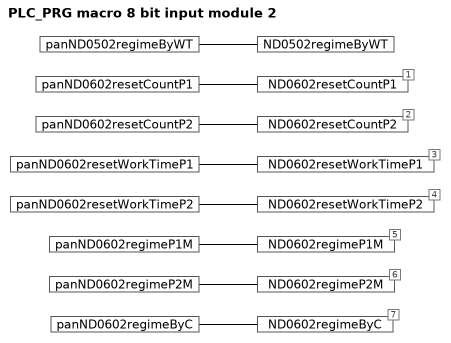
[picture p72: PLC_PRG macro 8 bit input module 2 (CFC)]
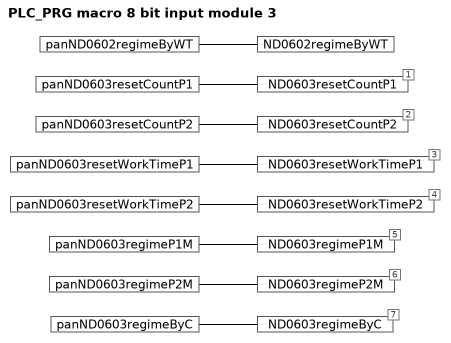
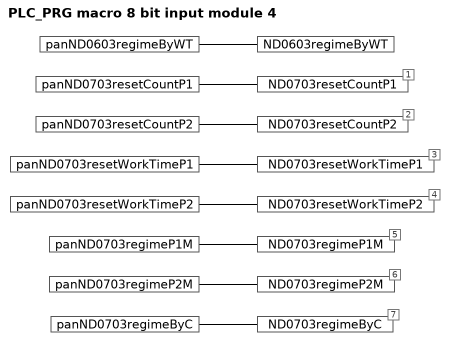
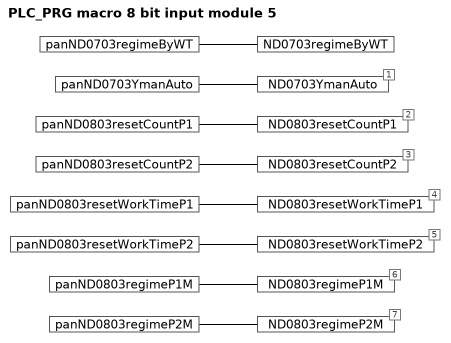
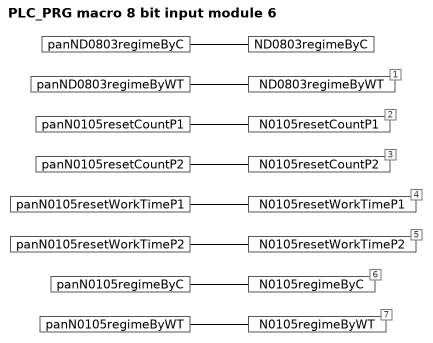
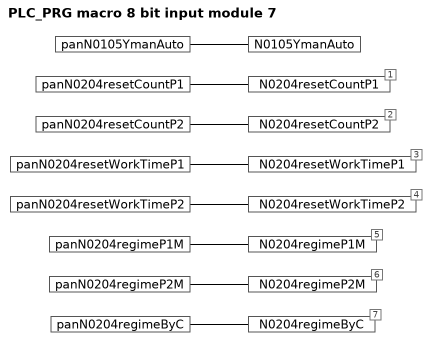
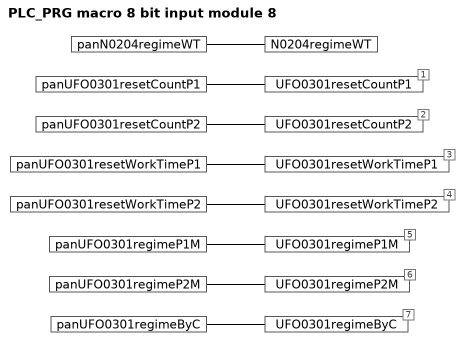
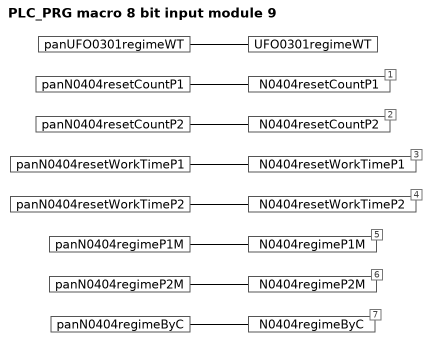
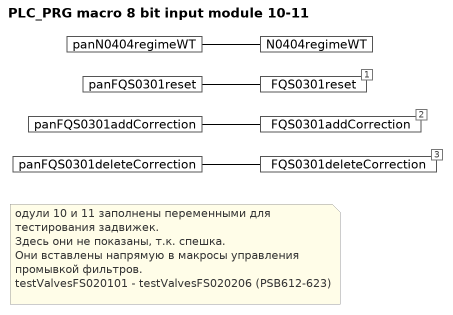
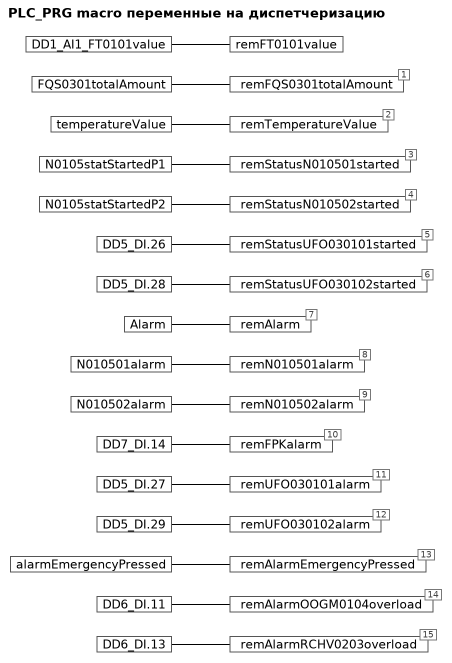
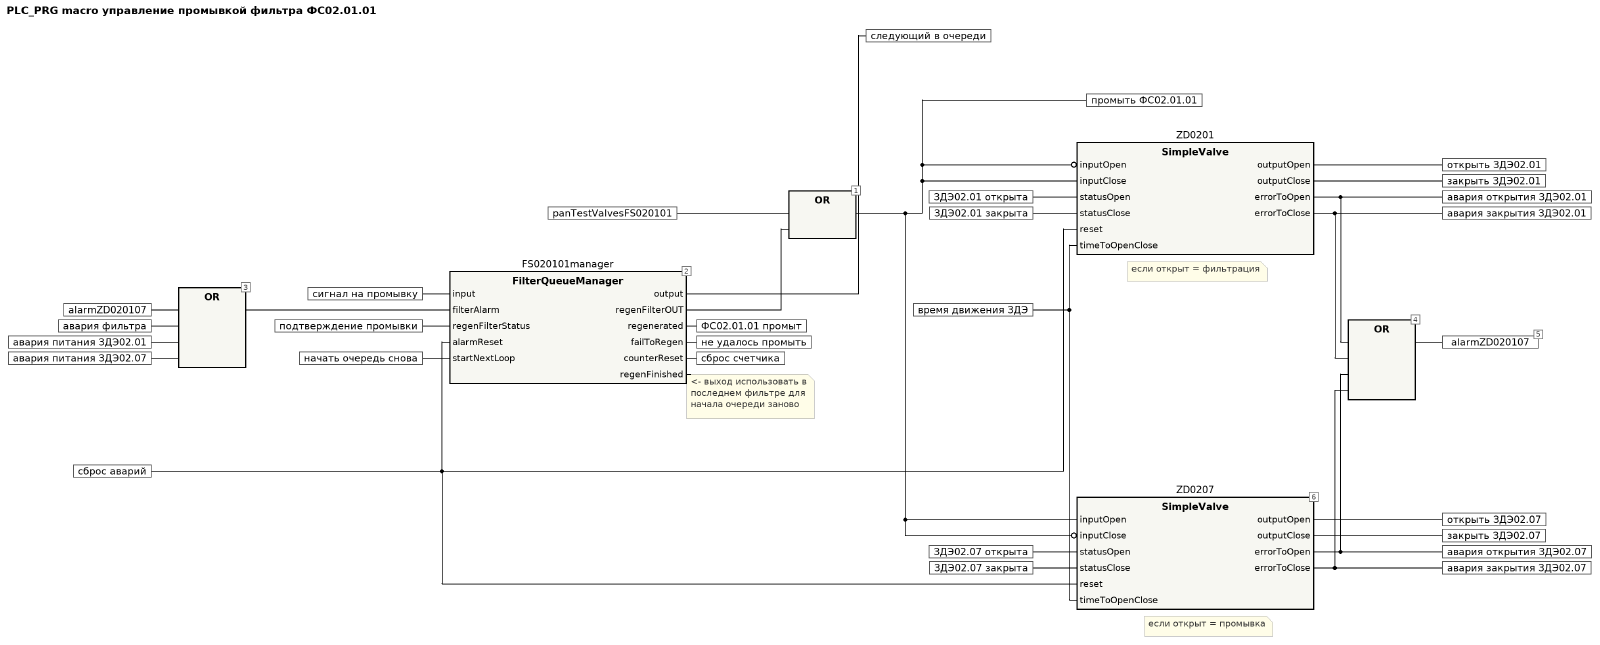
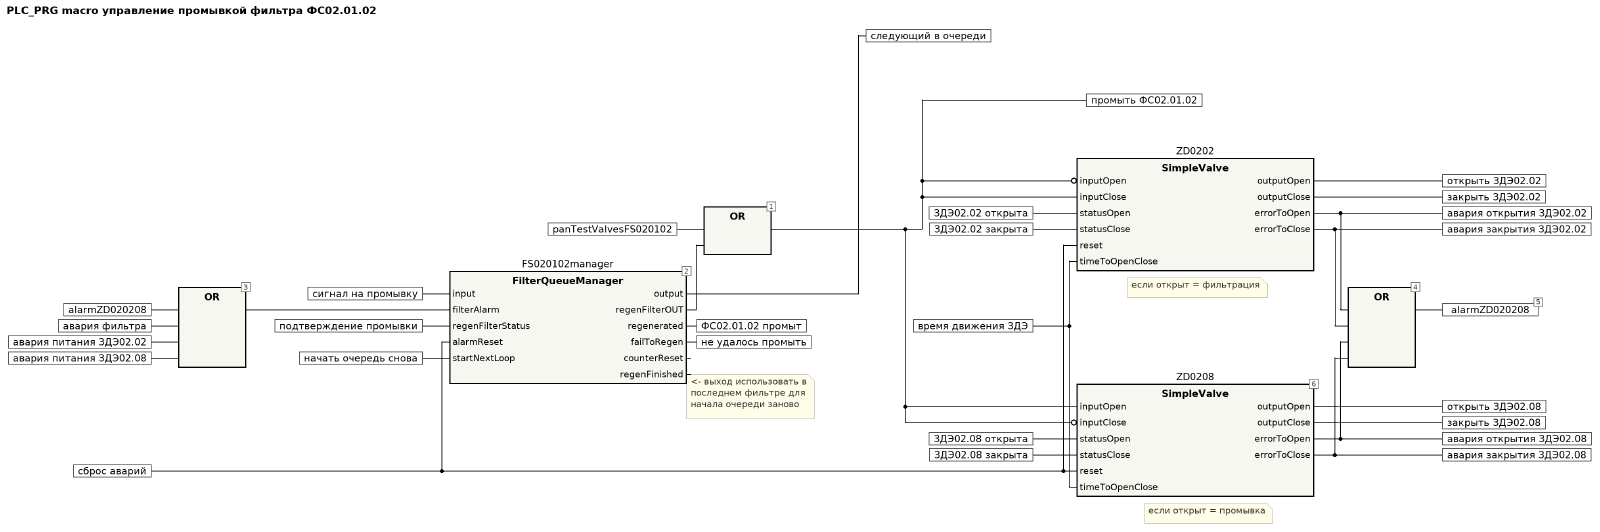
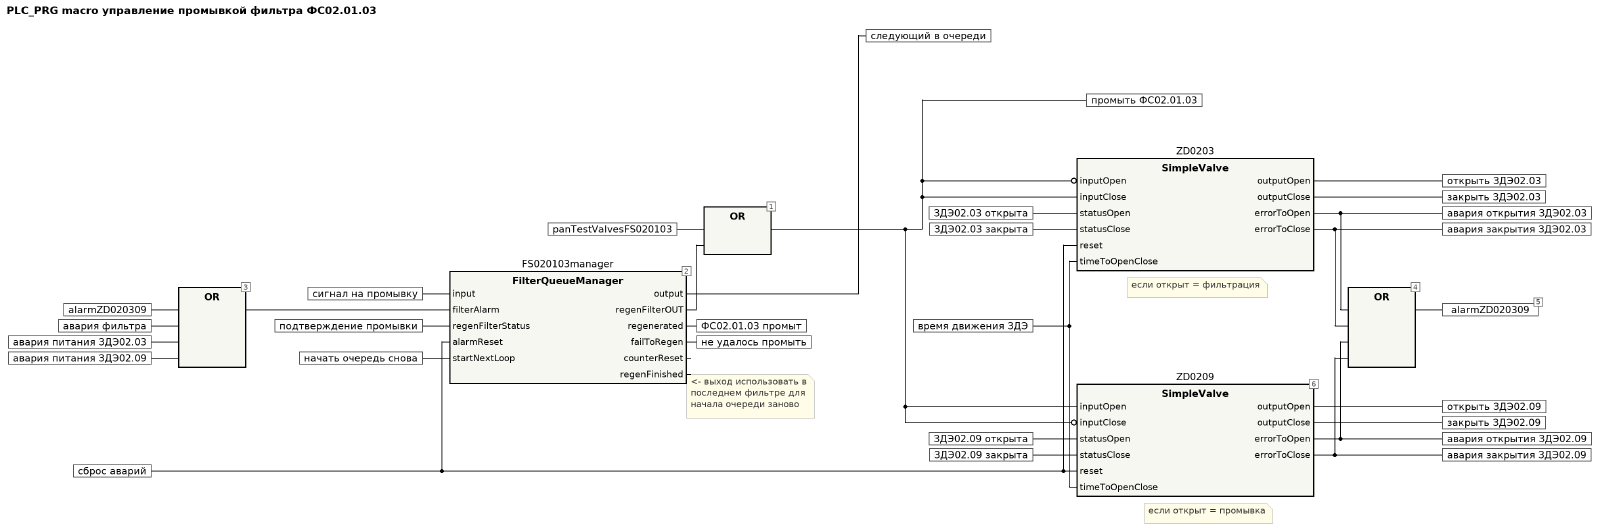
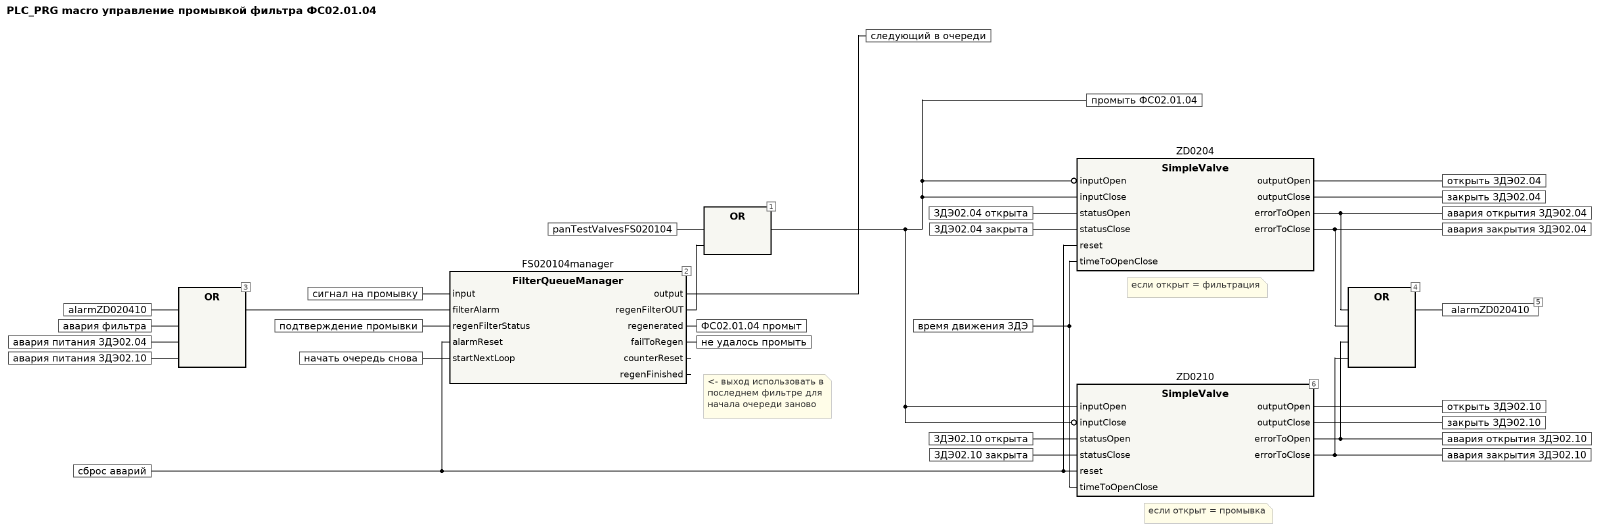
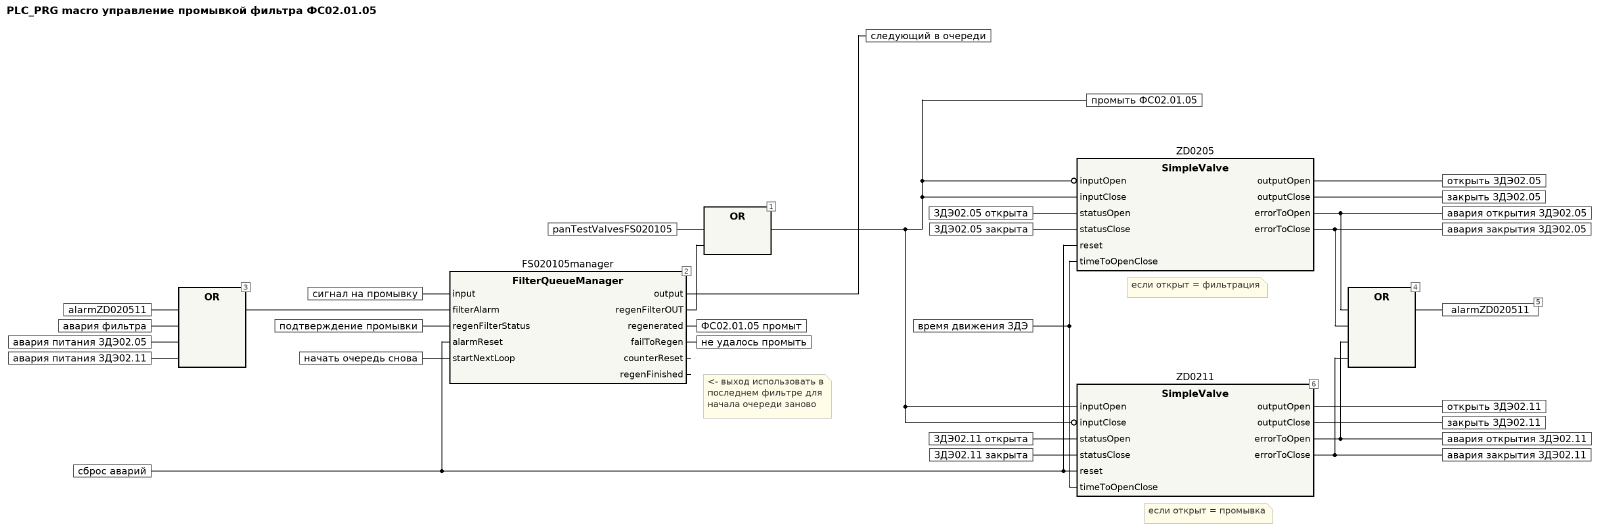
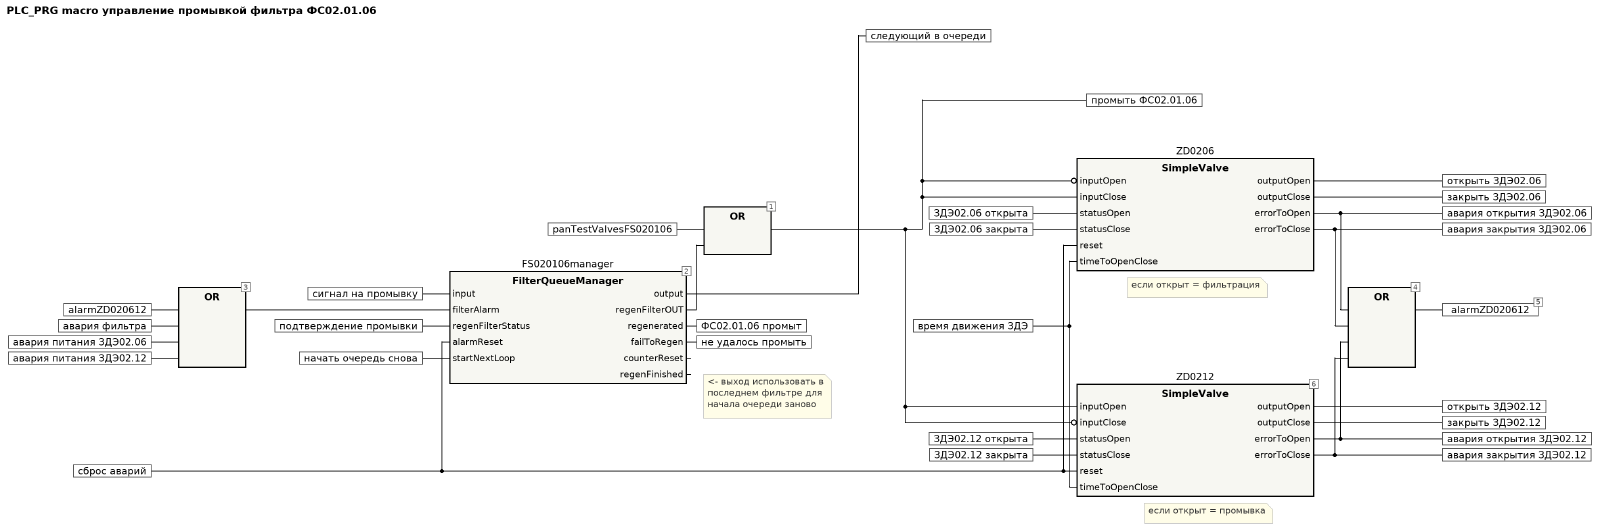
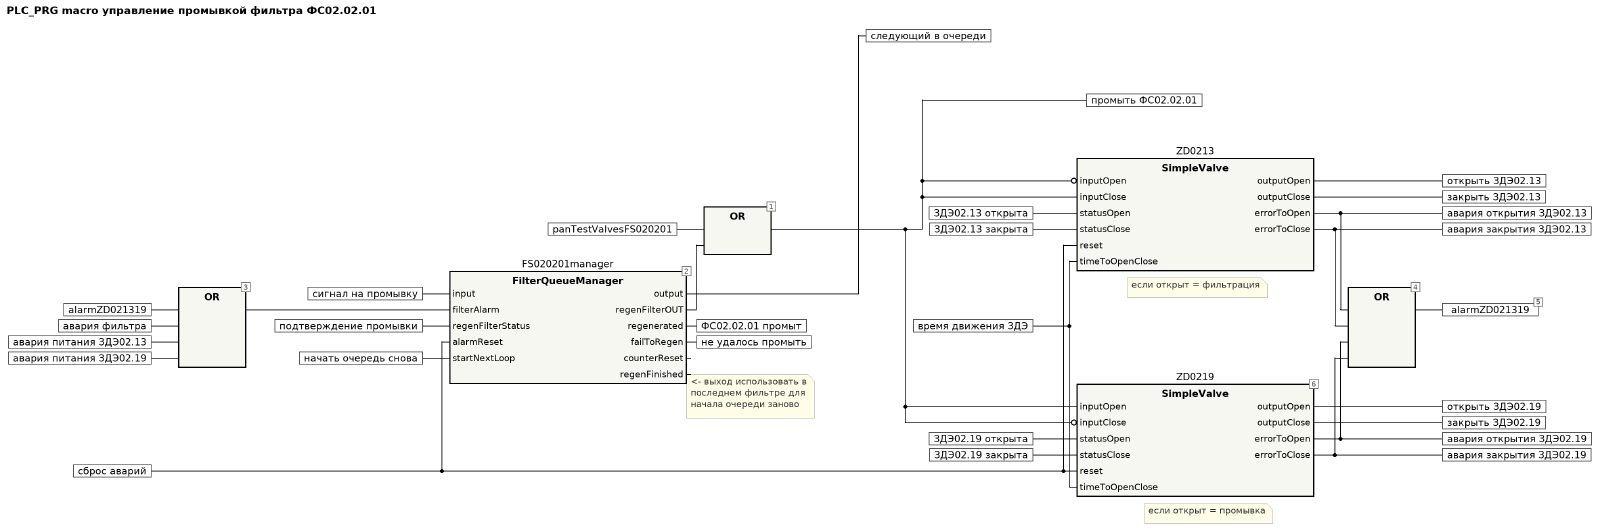
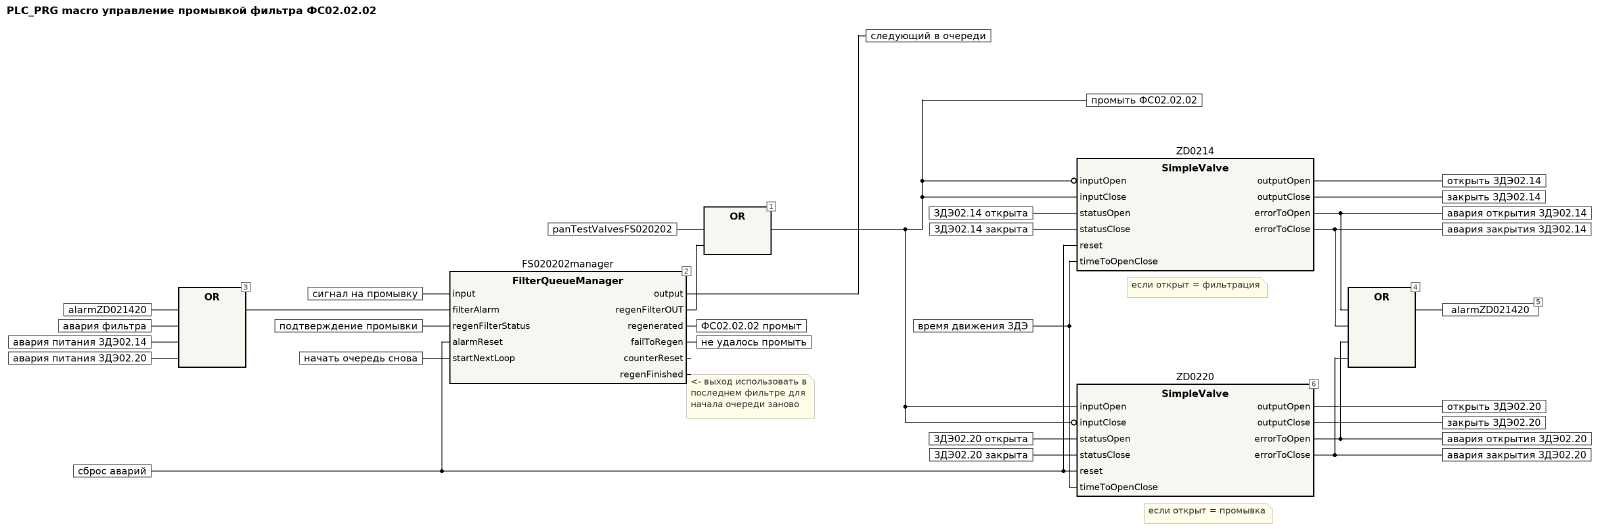
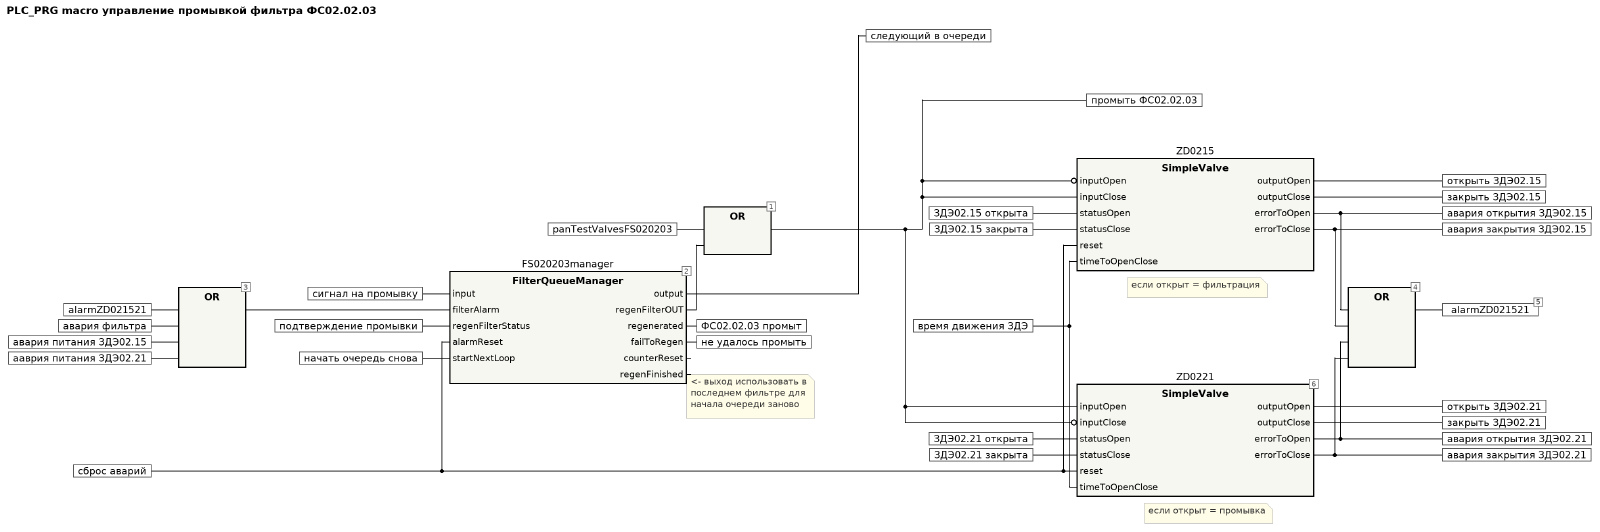
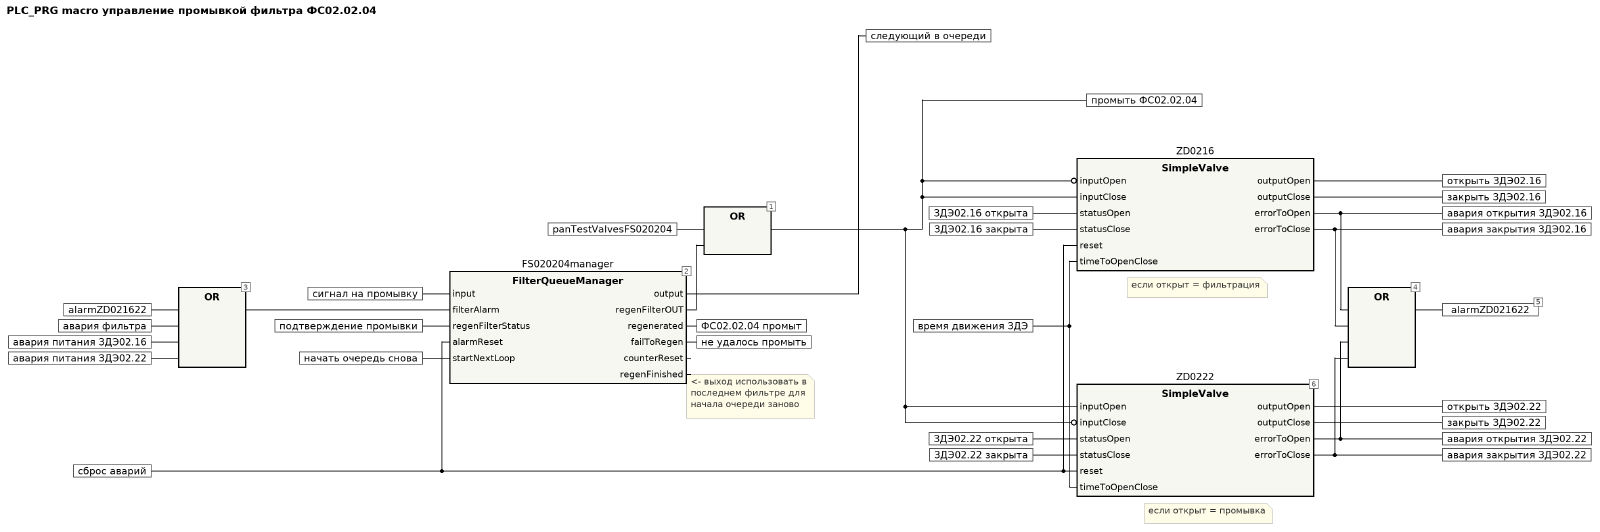
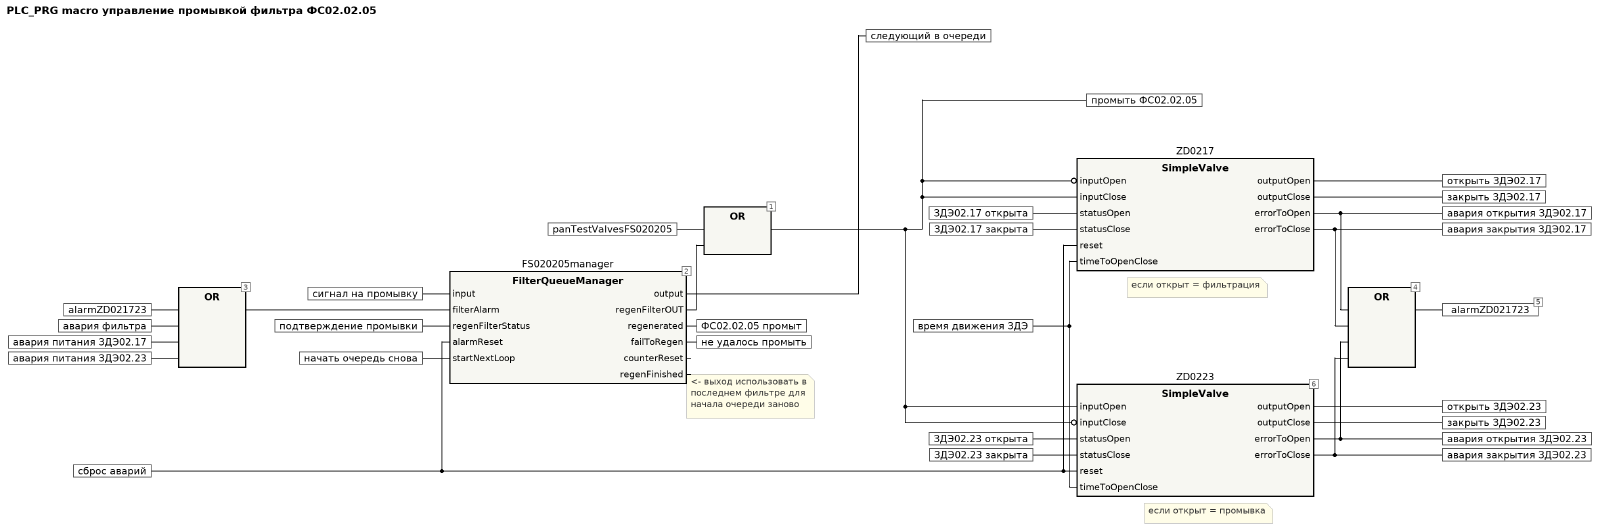
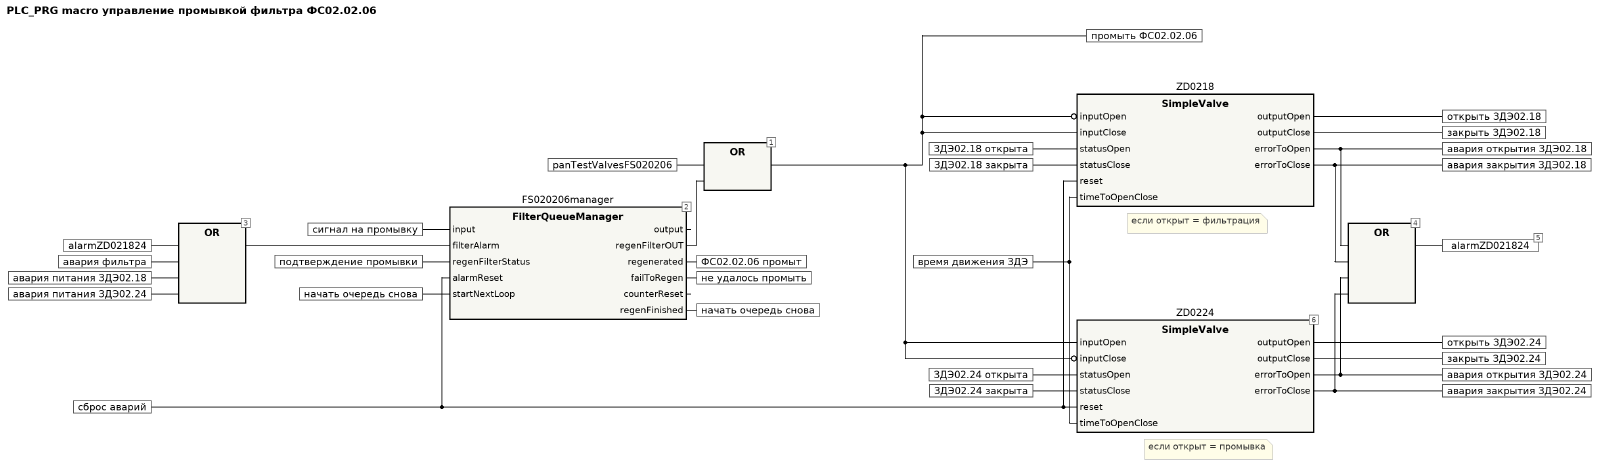
_CFC_ (* Continuous Function Chart, elements in execution order *)
(* 0 = перелив *)
(* авария обоих УФО, если проблемы / открытия/закрытия на одной из задвижек *)
(* авария питания ЗДЭ03.02 *)
(* авария питания ЗДЭ03.01 *)
(* статус-пуск Н01.05/02 *)
(* вкл КМ3 *)
(* Статус ПУСК / ЧРП Н01.05 *)
(* статус-пуск Н01.05/01 *)
(* вкл КМ2 *)
(* контроль обрыва или ошибок модулей в сети ПЛК *)
(* LSA01.02 перелив ОГМ01.04 *)
(* Нажат аварийный стоп. *)
(* авария сети (РКФ) *)
(* разрешение работы КНС / 1 = разрешено *)
(* Нажат аварийный стоп. *)
(* Блок управления разрешением работы КНС *)
(* авария сети (РКФ) *)
(* Авария питания клапанов КЭМ. *)
(* Авария питания розеток / управл.клапанов фильтров. *)
(* авария КНС *)
(* блок подачи сигнала на промывку *)
(* суммируем каждую секунду значение / мгновенного расхода в кубометрах в секунду *)
(* преобразуем расход из / кубометров в час в / кубометры в секунду *)
(* если есть расход / (больше нуля) *)
(* выдает импульс / каждую секунду *)
(* здесь мгновенный расход / в кубометрах в час (FT01.02) *)
(* Авария Н02.04/01 (0=авария) *)
(* Авария Н02.04/02 (0=авария) *)
(* промывка ФС02.01/06 *)
(* промывка ФС02.01/05 *)
(* промывка ФС02.01/04 *)
(* промывка ФС02.01/03 *)
(* промывка ФС02.01/02 *)
(* промывка ФС02.01/01 *)
(* пуск/стоп НД08.03/01 *)
(* пуск/стоп НД08.03/02 *)
(* пуск/стоп НД06.03/01 *)
(* пуск/стоп НД06.03/02 *)
(* пуск/стоп НД06.02/01 *)
(* пуск/стоп НД06.02/02 *)
(* пуск/стоп НД08.04 *)
(* пуск/стоп НД07.03/01 *)
(* пуск/стоп НД07.03/02 *)
(* авария М08.02 (УПФ) *)
(* авария М07.02 (УПЩ) *)
(* авария М06.04 (УПК) *)
(* работа М08.02 (УПФ) *)
(* работа М07.02 (УПЩ) *)
(* работа М06.04 (УПК) *)
(* Контроль, если УФО включили вручную, / а потока при этом нет. *)
(* авария УФО03.01/02 *)
(* работа УФО03.01/02 *)
(* авария УФО03.01/01 *)
(* Для подачи предостережения на пульте / оператора (при необходимости), а также / сигнализации лампой АВАРИЯ. *)
(* работа УФО03.01/01 *)
(* авария УФО03.01/02 *)
(* авария УФО03.01/01 *)
(* авария Н04.04/01 *)
(* авария Н04.04/02 *)
(* время контроля старта ФПК (по умолч.=3мин) *)
(* время работы ФПК после спада сигнала датч.осадка *)
(* запуск фильтрации *)
(* Защита от сухого хода насоса ФПК *)
(* датчик уровня осадка *)
(* Давление на входе ФПК (0...16 бар) *)
(* авария ФПК *)
(* подающий насос ФПК работает *)
(* ФПК готов к приему *)
(* ФПК не запустился *)
(* рН-метр QE01.02 на входе, / диапазон 0...14 *)
(* авария входа рН-метра QE01.01 *)
(* авария входа расходомера FT01.02 *)
(* расходомер FT01.01 на входе, / диапазон 0...600куб/час *)
(* авария НД08.04 *)
(* управление 4...20мА НД08.03/01 *)
(* пуск/стоп НД08.03/01 *)
(* пуск/стоп НД08.03/02 *)
(* управление 4...20мА НД08.03/02 *)
(* авария привода НД08.03/01 *)
(* авария привода НД08.03/02 *)
(* авария НД07.03/01 *)
(* авария НД07.03/02 *)
(* управление 4...20мА НД07.03/01 *)
(* управление 4...20мА НД07.03/02 *)
(* пуск/стоп НД07.03/01 *)
(* пуск/стоп НД07.03/02 *)
(* авария НД07.03/01 *)
(* авария НД07.03/02 *)
(* авария НД06.03/01 *)
(* авария НД06.03/02 *)
(* авария НД06.02/01 *)
(* авария НД06.02/02 *)
(* управление 4...20мА НД06.03/01 *)
(* пуск/стоп НД06.03/01 *)
(* пуск/стоп НД06.03/02 *)
(* управление 4...20мА НД06.03/02 *)
(* авария НД06.03/01 *)
(* авария НД06.03/02 *)
(* управление 4...20мА НД06.02/01 *)
(* пуск/стоп НД06.02/01 *)
(* пуск/стоп НД06.02/02 *)
(* управление 4...20мА НД06.02/02 *)
(* авария НД06.02/01 *)
(* авария НД06.02/02 *)
(* ошибка блока дозирования НД05.02 *)
(* авария входа датчика температуры *)
(* лампа АВАРИЯ *)
(* датчик температуры в помещении / (метран) диапазон: 0...+100С *)
(* управление 4...20мА НД05.02/01 *)
(* пуск/стоп НД05.02/01 *)
(* авария НД05.02/01 *)
(* авария НД05.02/02 *)
(* пуск/стоп НД05.02/02 *)
(* управление 4...20мА НД05.02/02 *)
(* АВАРИИ *)
(* авария привода НД08.03/01 *)
(* авария привода НД08.03/02 *)
(* авария НД08.04 *)
(* насос Н04.01 работает *)
(* пуск/стоп НД08.04 *)
(* управление 4...20мА НД08.04 *)
(* авария входа расходомера FT01.01 *)
(* расходомер FT01.02 на входе, / диапазон 0...600куб/час *)
(* рН-метр QE01.01 на входе, / диапазон 0...14 *)
(* авария входа рН-метра QE01.02 *)
(* сухой ход НД08.03/01 *)
(* сухой ход НД08.03/02 *)
(* сухой ход НД08.03/01 *)
(* сухой ход НД08.03/02 *)
(* LSA01.02 перелив ОГМ01.04 *)
(* Инициализирует требуемые булевые переменные / в момент старта выполнения программы. *)
(* Статус ПУСК ЧРП Н01.05 *)
(* LS01.03 - рабочий верхний уровень ОГМ01.04 автоматический пуск 01.05 *)
(* LS01.04 - нижний уровень ОГМ01.04, сухой ход Н01.05 *)
(* SA1 Ручной выбор Н01.05/01 = главный *)
(* SA1 Ручной выбор Н01.05/02 = главный *)
(* Стоп  Н01.05 (сброс самоподхвата реле) *)
(* время на создание потока *)
(* Пуск  Н01.05 *)
(* КМ1 питание ЧРП *)
(* КМ2 питание насоса 1 *)
(* КМ3 питание насоса 2 *)
(* Авария ЧРП Н01.05 *)
(* термоконтакт Н01.05/01 *)
(* термоконтакт Н01.05/02 *)
(* авария питания ЗДЭ02.25 *)
(* LSА02.01 Перелив РЧВ02.03 *)
(* Давление на входе ФПК / 0...16 бар (мах допуст.10) *)
(* Авария входа AI6 ПЛК, давл.ФПК *)
(* авария ФПК *)
(* Открыть КШЭ04.01 *)
(* статус КШЭ04.01 открыт *)
(* Закрыть КШЭ04.01 *)
(* статус КШЭ04.01 закрыт *)
(* подающий насос ФПК работает *)
(* стоп Н04.04 *)
(* пуск Н04.04/02 *)
(* пуск Н04.04/01 *)
(* авт.пуск Н04.04 *)
(* сухой ход Н04.04, 0=защита *)
(* авария Н04.04/01, 0=авария *)
(* авария Н04.04/02, 0=авария *)
(* импульсный расходомер *)
(* Авария Н02.04/01 (0=авария) *)
(* Авария Н02.04/02 (0=авария) *)
(* промывка ФС02.02/06 *)
(* промывка ФС02.02/05 *)
(* промывка ФС02.02/04 *)
(* промывка ФС02.02/03 *)
(* промывка ФС02.02/02 *)
(* промывка ФС02.02/01 *)
(* Клапан КЭМ05.01 открыт. *)
(* Клапан КЭМ06.01 открыт. *)
(* Клапан КЭМ07.01 открыт. *)
(* Клапан КЭМ08.01 открыт. *)
(* Сухой ход Н02.04 (LS02.03) 0=сух.ход *)
(* Стоп Н02.04 *)
(* Пуск Н02.04/01 *)
(* Пуск Н02.04/02 *)
(* текущий объем *)
(* заданный до промывки объем *)
(* 0=авария *)
(* авария (при 0) ФС02.01/06 *)
(* авария (при 0) ФС02.01/05 *)
(* авария (при 0) ФС02.01/04 *)
(* авария (при 0) ФС02.01/03 *)
(* авария (при 0) ФС02.01/02 *)
(* авария (при 0) ФС02.01/01 *)
(* авария (при 0) ФС02.02/06 *)
(* авария (при 0) ФС02.02/05 *)
(* авария (при 0) ФС02.02/04 *)
(* авария (при 0) ФС02.02/03 *)
(* авария (при 0) ФС02.02/02 *)
(* авария (при 0) ФС02.02/01 *)
(* сброс счетчика стоков до следующей промывки *)
(* подсчет общего объема стоков, прошедшего через расходомер FT01.02 *)
(* очередь передается на 2 ступень *)
(* авария питания ЗДЭ02.01 *)
(* авария питания ЗДЭ02.02 *)
(* авария питания ЗДЭ02.03 *)
(* авария питания ЗДЭ02.04 *)
(* авария питания ЗДЭ02.05 *)
(* авария питания ЗДЭ02.06 *)
(* авария питания ЗДЭ02.07 *)
(* авария питания ЗДЭ02.08 *)
(* авария питания ЗДЭ02.09 *)
(* авария питания ЗДЭ02.10 *)
(* авария питания ЗДЭ02.11 *)
(* авария питания ЗДЭ02.12 *)
(* авария питания ЗДЭ02.13 *)
(* авария питания ЗДЭ02.14 *)
(* авария питания ЗДЭ02.15 *)
(* авария питания ЗДЭ02.16 *)
(* авария питания ЗДЭ02.17 *)
(* авария питания ЗДЭ02.18 *)
(* авария питания ЗДЭ02.19 *)
(* авария питания ЗДЭ02.20 *)
(* авария питания ЗДЭ02.21 *)
(* авария питания ЗДЭ02.22 *)
(* авария питания ЗДЭ02.23 *)
(* авария питания ЗДЭ02.24 *)
(* инвертирование сигнала, чтобы все аварии / обозначались как 1 (TRUE) *)
(* авария НД05.02/01 *)
(* авария НД05.02/02 *)
(* авария питания КШЭ04.01 *)
(* 1=открыть; 0 = закрыть *)
(* в этом макросе лежит управление режимом тестирования задвижек ЗДЭ03 / Тестирование запрещает автоматический запуск УФО от ПЛК *)
#0 rTrigStartInitializer:R_TRIG(CLK: TRUE)
#1 startInitializer <= #0.Q
#2 MACRO контроль температуры в помещении(pin 1 "вход датчика температуры": DD1_AI0, pin 2 "минимально допустимая температура в помещении": maxTemperature, pin 3 "максимально допустимая температура в помещении": minTemperature)
	(* задаем границы допустимой температуры в помещении / проверяем что измеренное значение в заданном диапазоне *)
	(* не смотрим конкретный тип ошибки / (работает не точно, обрыв определяет как слишком маленькое значение) / если не равно 0 - значит на входе ошибка *)
	#3 DD1_AI0_temperature:DECODE_FLOAT(VALUE: pin 1, DEF_VALUE: -)
	#4 NE(#3._ERR, 0)
	out 2 "авария датчика температуры" <= #4
	out 1 "температура в помещении" <= #3.OUT_VALUE
	#5 REAL_TO_INT(#3.OUT_VALUE)
	#6 temperatureLimits:LIMITALARM(IN: #5, HIGH: pin 3, LOW: pin 2)
	out 3 "температура выше заданного диапазона" <= #6.O
	out 4 "температура ниже заданного диапазона" <= #6.U
	#7 temperatureLimits:LIMITALARM(IN: -, HIGH: -, LOW: -)
END_MACRO
#8 temperatureValue <= #2.out 1
#9 DD1_AI0_error <= #2.out 2
#10 alarmHighTemperature <= #2.out 3
#11 alarmLowTemperature <= #2.out 4
#12 OR(testKSHE0401, DD7_DI.13)
#13 MACRO клапан шаровый перед ФПК (КШЭ04.01)(pin 1 "сигнал "подающий насос ФПК" работает": #12, pin 2 "статус КШЭ04.01 открыт": DD9_DI.2, pin 3 "статус КШЭ04.01 закрыт": DD9_DI.3, pin 4 "сброс аварий": alarmReset, pin 5 "время на открытие/закрытие": timeToOpenCloseValve)
	#14 FPKkshe0401DelayToOpen:TON(IN: #16.outputOpen, PT: T#1s)
	out 1 "выход на открытие КШЭ04.01" <= #14.Q
	#15 FPKkshe0401DelayToClose:TON(IN: #16.outputClose, PT: T#1s)
	out 2 "выход на закрытие КШЭ04.01" <= #15.Q
	#16 FPKkshe0401:SimpleValve(inputOpen: pin 1, inputClose: #17, statusOpen: pin 2, statusClose: pin 3, reset: pin 4, timeToOpenClose: pin 5)
	#17 NOT(pin 1)
	out 3 "авария на открытие КШЭ04.01" <= #16.errorToOpen
	out 4 "авария на закрытие КШЭ04.01" <= #16.errorToClose
END_MACRO
#18 DD4_DO.2 <= #13.out 1
#19 DD4_DO.3 <= #13.out 2
#20 FPKkshe0401errorToOpen <= #13.out 3
#21 FPKkshe0401errorToClose <= #13.out 4
#22 OR(DD1_AI0_error, DD1_AI1_error, DD1_AI2_error, DD1_AI3_error, DD1_AI4_error, alarmHighTemperature, alarmLowTemperature, ND0502dosingError, ND0602dosingError, ND0603dosingError, ND0803dosingError, ND0804dosingError, DD1_DI6, DD1_DI7, N010501alarm, N010502alarm, ZDE0225errorToOpen, ZDE0225errorToClose, DD7_DI.14, FPKnotStarted, DD1_AI5_error, FPKkshe0401errorToOpen, FPKkshe0401errorToClose, DD5_DI.27, DD5_DI.29, filterFailToRegen020101, errorToOpenZD0201, errorToCloseZD0201, errorToOpenZD0207, errorToCloseZD0207, filterFailToRegen020102, errorToOpenZD0202, errorToCloseZD0202, errorToOpenZD0208, errorToCloseZD0208, filterFailToRegen020103, errorToOpenZD0203, errorToCloseZD0203, errorToOpenZD0209, errorToCloseZD0209, filterFailToRegen020104, errorToOpenZD0204, errorToCloseZD0204, errorToOpenZD0210, errorToCloseZD0210, filterFailToRegen020105, errorToOpenZD0205, errorToCloseZD0205, errorToOpenZD0211, errorToCloseZD0211, filterFailToRegen020106, errorToOpenZD0206, errorToCloseZD0206, errorToOpenZD0212, errorToCloseZD0212, filterFailToRegen020201, errorToOpenZD0213, errorToCloseZD0213, errorToOpenZD0219, errorToCloseZD0219, filterFailToRegen020202, errorToOpenZD0214, errorToCloseZD0214, errorToOpenZD0220, errorToCloseZD0220, filterFailToRegen020203, errorToOpenZD0215, errorToCloseZD0215, errorToOpenZD0221, errorToCloseZD0221, filterFailToRegen020204, errorToOpenZD0216, errorToCloseZD0216, errorToOpenZD0222, errorToCloseZD0222, filterFailToRegen020205, errorToOpenZD0217, errorToCloseZD0217, errorToOpenZD0223, errorToCloseZD0223, filterFailToRegen020206, errorToOpenZD0218, errorToCloseZD0218, errorToOpenZD0224, errorToCloseZD0224, alarmPLKnetwork, alarmND050201, alarmND050202, alarmND060201, alarmND060202, alarmND060301, alarmND060302, alarmND070301, alarmND070302, alarmND080301, alarmND080302, alarmND0804, alarmOGM0104overload, alarmRCHV0203overload, alarmN040402, alarmN040401, alarmM0604, alarmM0702, alarmM0802, alarmN020401, alarmN020402, alarmFS020101, alarmFS020102, alarmFS020103, alarmFS020104, alarmFS020105, alarmFS020106, alarmFS020201, alarmFS020202, alarmFS020203, alarmFS020204, alarmFS020205, alarmFS020206, alarmZDE0201power, alarmZDE0202power, alarmZDE0203power, alarmZDE0204power, alarmZDE0205power, alarmZDE0206power, alarmZDE0207power, alarmZDE0208power, alarmZDE0209power, alarmZDE0210power, alarmZDE0211power, alarmZDE0212power, alarmZDE0213power, alarmZDE0214power, alarmZDE0215power, alarmZDE0216power, alarmZDE0217power, alarmZDE0218power, alarmZDE0219power, alarmZDE0220power, alarmZDE0221power, alarmZDE0222power, alarmZDE0223power, alarmZDE0224power, alarmZDE0225power, alarmKSHE0401power, alarmKNS, alarmPowerSocketFS, alarmKEMvalvesPower, alarmEmergencyPressed, alarmRKF, errorToOpenZDE0301, errorToCloseZDE0301, errorToOpenZDE0302, errorToCloseZDE0302, alarmZDE0301power, alarmZDE0302power)
#23 DD1_DO11 <= #22
#24 alarm <= #22
#25 MACRO контроль аналогового входа DD1_AI1(pin 1 "вход": DD1_AI1)
	(* Не смотрим конкретную ошибку, / определяем,что вход неисправен без расшифровки. *)
	#26 DD1_AI1_FT0101:DECODE_FLOAT(VALUE: pin 1, DEF_VALUE: -)
	#27 NE(#26._ERR, 0)
	out 2 "авария" <= #27
	out 1 "выход" <= #26.OUT_VALUE
END_MACRO
#28 DD1_AI1_FT0101value <= #25.out 1
#29 DD1_AI1_error <= #25.out 2
#30 MACRO контроль аналогового входа DD1_AI2(pin 1 "вход": DD1_AI2)
	(* Не смотрим конкретную ошибку, / определяем,что вход неисправен без расшифровки. *)
	#31 DD1_AI2_FT0102:DECODE_FLOAT(VALUE: pin 1, DEF_VALUE: -)
	#32 NE(#31._ERR, 0)
	out 2 "авария" <= #32
	out 1 "выход" <= #31.OUT_VALUE
END_MACRO
#33 DD1_AI2_FT0102value <= #30.out 1
#34 DD1_AI2_error <= #30.out 2
#35 MACRO управление Н01.05 (поддержание заданного расхода по FT01.02)(pin 1 "статус ПУСК ЧРП (реле)": DD5_DI.4, pin 2 "LS01.03 раб.уров.": DD6_DI.12, pin 3 "LS01.04 ниж.уров.(сух.ход)": DD5_DI.0, pin 4 "SA1ручной выб.Н01.05/01-главный": DD5_DI.5, pin 5 "SA1ручной выб.Н01.05/02-главный": DD5_DI.6, pin 6 "включить режим "по кол.вкл."": N0105regimeByC, pin 7 "включить режим "по наработке"": N0105regimeByWT, pin 8 "значение расхода от FT01.02": DD1_AI2_FT0102value, pin 9 "уставка расхода": N0105flowSetValue, pin 10 "время на создание потока": N0105minFlowTime, pin 11 "Р-коэфф.": N0105koeffP, pin 12 "I-коэфф": N0105koeffI, pin 13 "Д-коэфф": N0105koeffD, pin 14 "управление ЧРП в ручн.реж.(4...20мА)": N0105YoutManual, pin 15 "переключатель управление ЧРП РУЧН/АВТ": N0105YmanAuto, pin 16 "мин.допустимый расход": N0105minFlow, pin 17 "термоконтакт Н01.05/01": DD5_DI.2, pin 18 "термоконтакт Н01.05/02": DD5_DI.3, pin 19 "авария ЧРП Н01.05": DD5_DI.1, pin 20 "сброс аварии": alarmReset, pin 21 "сброс кол-ва вкл.Н01.05/01": N0105resetCountP1, pin 22 "сброс кол-ва вкл.Н01.05/02": N0105resetCountP2, pin 23 "сброс наработки Н01.05/01": N0105resetWorkTimeP1, pin 24 "сброс наработки Н01.05/02": N0105resetWorkTimeP2)
	(* время на создание потока *)
	(* Пуск  Н01.05 *)
	(* режимы по количеству включений,  или по наработке / активны если оба входа SA1 не активны *)
	(* управление Н01.05 - поддержание / заданного расхода по FT01.02 *)
	(* по умолчанию при старте программы *)
	(* если на входе true / то нижнее значение, / иначе то, что посередине *)
	(* Если насос создает давление меньше / указанного, то авария. *)
	#36 OR(pin 2, #37.Q)
	#37 N0105startTrig:R_TRIG(CLK: pin 1)
	#38 N0105stopTrig:F_TRIG(CLK: pin 1)
	#39 N0105startTrigg:RS(SET: #36, RESET1: #41)
	#40 N0105regime:choosePumpRegime(start: #39.Q1, pump1Main: pin 4, pump2Main: pin 5, byCounter: #44, byWorkTime: #50)
	out 2 "статус режим "Н01.05/01 - главный"" <= #40.pump1MainActive
	out 3 "статус режим "Н01.05/02 - главный"" <= #40.pump2MainActive
	out 4 "статус режим "по кол-ву вкл."" <= #40.byCounterActive
	#41 OR(#38.Q, #42)
	out 5 "статус режим "по наработке"." <= #40.byWorkTimeActive
	#42 NOT(pin 3)
	#43 NOT(#39.Q1)
	out 1 "СТОП (сброс самоподхвата реле пуска ЧРП)." <= #43
	#44 AND(NOT pin 4, NOT pin 5, #47.Q1)
	#45 OR(pin 6, startInitializer)
	#46 N0105regByCinit:R_TRIG(CLK: #45)
	#47 N0105regByCtrig:RS(SET: #46.Q, RESET1: #55.Q)
	#48 N0105twoPumpOneDriveManager:TwoPumpOneDriveManager(startStopPump1: #40.startPump1, startStopPump2: #40.startPump2, alarmPump1: N010501alarm, alarmPump2: N010502alarm, alarmReset: alarmReset, counterStart: #40.startByCounter, Pump1ResetCounter: pin 21, Pump2ResetCounter: pin 22, ValueToResetCounter: -, workTimeStart: #40.startByWorkTime, workTimePump1Reset: pin 23, workTimePump2Reset: pin 24, timeKM1off: -, timeKM23DelayON: -, timeKM23offDelay: -, timeReadyToStartDelay: -)
	out 6 "кол-во включений Н01.05/01" <= #48.counterPump1
	#49 AND(#48.pump1active, #65)
	out 7 "кол-во включений Н01.05/02" <= #48.counterPump2
	out 8 "наработка Н01.05/01" <= #48.currentWorkTimePump1
	out 15 "авария Н01.05/01" <= #53.Q1
	#50 AND(NOT pin 4, NOT pin 5, #56.Q1)
	out 9 "наработка Н01.05/02" <= #48.currentWorkTimePump2
	out 10 "КМ1-питание ЧРП" <= #48.DriveKM
	#51 AND(#48.pump1active, #57)
	#52 OR(#49, #51)
	#53 N010501alarmTrig:RS(SET: #52, RESET1: pin 20)
	#54 N010501alarm <= #53.Q1
	#55 N0105regWTinit:R_TRIG(CLK: pin 7)
	#56 N0105regWTtrig:RS(SET: #55.Q, RESET1: #46.Q)
	out 11 "КМ2-питание Н01.05/01" <= #48.pump1KM
	out 12 "КМ3-питание Н01.05/02" <= #48.pump2KM
	#57 OR(NOT pin 17, NOT pin 19)
	out 13 "пуск ЧРП (Н01.05)" <= #48.driveStart
	#58 OR(NOT pin 19, NOT pin 18)
	out 16 "авария Н01.05/02" <= #61.Q1
	#59 AND(#58, #48.pump2active)
	#60 OR(#59, #63)
	#61 N010502alarmTrig:RS(SET: #60, RESET1: pin 20)
	#62 N010502alarm <= #61.Q1
	#63 AND(#48.pump2active, #65)
	#64 N0105timerminFlow:TON(IN: #48.driveStart, PT: pin 10)
	#65 AND(#64.Q, #66)
	#66 LE(pin 8, pin 16)
	#67 SEL(#48.driveStart, 0, #68.Y)
	out 14 "управление ЧРП (4...20мА)" <= #67
	#68 N0105pidReg:PID(ACTUAL: pin 8, SET_POINT: pin 9, KP: pin 11, TN: pin 12, TV: pin 13, Y_MANUAL: pin 14, Y_OFFSET: -, Y_MIN: 4, Y_MAX: 20, MANUAL: pin 15, RESET: #68.OVERFLOW)
END_MACRO
#69 DD4_DO.13 <= #35.out 1
#70 N0105statRegimeP1M <= #35.out 2
#71 N0105statRegimeP2M <= #35.out 3
#72 N0105statRegimeByC <= #35.out 4
#73 N0105statRegimeByWT <= #35.out 5
#74 N0105counterP1 <= #35.out 6
#75 N0105counterP2 <= #35.out 7
#76 N0105workTimeP1 <= #35.out 8
#77 N0105workTimeP2 <= #35.out 9
#78 DD2_DO.0 <= #35.out 10
#79 DD2_DO.1 <= #35.out 11
#80 DD2_DO.2 <= #35.out 12
#81 DD1_DO0 <= #35.out 13
#82 DD1_AO0 <= #35.out 14
#83 N010501alarm <= #35.out 15
#84 N010502alarm <= #35.out 16
#85 MACRO Сигналы работы с ФП04.02 (фильтр-пресс)(pin 1 "датчик уровня осадка": DD7_DI.15, pin 2 "время работы ФПК (после выкл.датч.осадка)": FPKtimeToWork, pin 3 "защита от сухого хода": DD6_DI.10, pin 4 "ошибка входа AI (обрыв)": DD1_AI5_error, pin 5 "авария ФПК": DD7_DI.14, pin 6 "фильтр-пресс готов к приему": DD7_DI.12, pin 7 "давление на входе в ФПК": DD1_AI5_FPKpressureValue, pin 8 "мах допустимое давление": FPKmaxPressureValue, pin 9 "подающий насос ФПК работает": DD7_DI.13, pin 10 "время контроля старта ФПК": FPKnotStartedTime, pin 11 "сброс аварий": alarmReset)
	(* ФПК готов к приему осадка *)
	(* LS01.01-нижн.уровень на входе ОГМ01.04 / защита от сух. хода насоса ФПК *)
	(* LES01.01-сигнал датчика уровня осадка ОГМ01.04 / запуск процесса фильтрации *)
	(* Время работы ФПК после / спада сигнала уровня осадка / по умолч.15мин. *)
	(* Давление на входе ФПК / 0...16 бар (мах допуст.10) *)
	(* максимально допустимое давление / на входе ФПК *)
	(* Условие сброса сигнала о грязном фильтр-прессе: / 1. Пропал сигнал о готовности ФПК; / 2. Появился сигнал о готовности ФПК. / Это значит, что оператор раздвигал плиты, / чистил и снова сдвигал их. *)
	#86 FPKneedToCleanResetFtrig:F_TRIG(CLK: FPKneedToCleanReset)
	#87 FPKstartTrig:RS(SET: pin 1, RESET1: #93)
	out 1 "запуск/старт ФПК" <= #87.Q1
	#88 FPKstopTimer:TOF(IN: pin 1, PT: pin 2)
	#89 FPKstopFtrig:F_TRIG(CLK: #88.Q)
	#90 AND(#87.Q1, #91)
	#91 NOT(pin 11)
	#92 AND(#87.Q1, #94.Q, #96)
	out 2 "ФПК не стартовал" <= #92
	#93 OR(#89.Q, pin 4, pin 5, #95, #97, #100.Q1)
	#94 FPKnotStartedTimer:TON(IN: #90, PT: pin 10)
	#95 NOT(pin 3)
	#96 NOT(pin 9)
	#97 NOT(pin 6)
	#98 AND(#87.Q1, #99)
	#99 GE(pin 7, pin 8)
	#100 FPKneedToCleanTrig:RS(SET: #98, RESET1: #86.Q)
	out 3 "ФПК нужно почистить!" <= #100.Q1
	#101 S FPKneedToCleanReset <= #100.Q1
	#102 FPKneedToCleanResetRtrig:R_TRIG(CLK: pin 6)
	#103 R FPKneedToCleanReset <= #102.Q
END_MACRO
#104 DD1_DO10 <= #85.out 1
#105 FPKnotStarted <= #85.out 2
#106 FPKneedToClean <= #85.out 3
#107 MACRO контроль аналогового входа DD1_AI3(pin 1 "вход": DD1_AI3)
	(* Не смотрим конкретную ошибку, / определяем,что вход неисправен без расшифровки. *)
	#108 DD1_AI3_QE0101:DECODE_FLOAT(VALUE: pin 1, DEF_VALUE: -)
	#109 NE(#108._ERR, 0)
	out 2 "авария" <= #109
	out 1 "выход" <= #108.OUT_VALUE
END_MACRO
#110 DD1_AI3_QE0101value <= #107.out 1
#111 DD1_AI3_error <= #107.out 2
#112 MACRO контроль аналогового входа DD1_AI4(pin 1 "вход": DD1_AI4)
	(* Не смотрим конкретную ошибку, / определяем,что вход неисправен без расшифровки. *)
	#113 DD1_AI4_QE0102:DECODE_FLOAT(VALUE: pin 1, DEF_VALUE: -)
	#114 NE(#113._ERR, 0)
	out 2 "авария" <= #114
	out 1 "выход" <= #113.OUT_VALUE
END_MACRO
#115 DD1_AI4_QE0102value <= #112.out 1
#116 DD1_AI4_error <= #112.out 2
#117 MACRO контроль аналогового входа DD1_AI5(pin 1 "вход": DD1_AI5)
	(* Не смотрим конкретную ошибку, / определяем,что вход неисправен без расшифровки. *)
	#118 DD1_AI5_FPK:DECODE_FLOAT(VALUE: pin 1, DEF_VALUE: -)
	#119 NE(#118._ERR, 0)
	out 2 "авария" <= #119
	out 1 "выход" <= #118.OUT_VALUE
END_MACRO
#120 DD1_AI5_FPKpressureValue <= #117.out 1
#121 DD1_AI5_error <= #117.out 2
#122 MACRO управление НД05.02 УПГ(pin 1 "вход расходомера в куб/час": DD1_AI1_FT0101value, pin 2 "max производительность НД в мл/мин": ND0502setMaxDosVal, pin 3 "задание дозирования в мл/куб": ND0502setKoefProp, pin 4 "режим:1 насос главный": ND0502regimeP1M, pin 5 "режим: 2 насос главный": ND0502regimeP2M, pin 6 "режим: по наработке": ND0502regimeByWT, pin 7 "режим: по кол-ву включений": ND0502regimeByC, pin 8 "авария 1 насоса": DD6_DI.0, pin 9 "авария 2 насоса": DD6_DI.1, pin 10 "сброс аварий": alarmReset, pin 11 "сброс счетчика включений 1 насоса": ND0502resetCountP1, pin 12 "сброс ссчетчика включений 2 насоса": ND0502resetCountP2, pin 13 "сброс наработки 1 насоса": ND0502resetWorkTimeP1, pin 14 "сброс наработки 2 насоса": ND0502resetWorkTimeP2)
	(* сигнал 4...20мА на НД05.02/02 *)
	(* сигнал 4...20мА на НД05.02/01 *)
	(* Если на входе SEL = TRUE, / то нижнее значение, / иначе - то,что посередине. *)
	#123 SEL(#129.pump1ON, 0, #124.outputValue)
	out 6 "выход 4...20мА насоса 1" <= #123
	#124 ND0502dosing:DosingPumpProportional(flowValue: pin 1, setMinPumpDosingValue: -, setMaxPumpDosingValue: pin 2, minOutputValue: -, maxOutputValue: -, setKoeffProportionality: pin 3, minFlowToStart: -)
	out 1 "ошибка блока дозирования" <= #124.dosingError
	#125 SEL(#129.pump2ON, 0, #124.outputValue)
	#126 REAL_TO_WORD(#125)
	out 7 "выход 4...20мА насоса 2" <= #126
	#127 ND0502regime:choosePumpRegime(start: #124.startDosingPump, pump1Main: pin 4, pump2Main: pin 5, byCounter: #128, byWorkTime: pin 6)
	out 2 "статус: 1 насос главный" <= #127.pump1MainActive
	out 3 "статус: 2 насос главный" <= #127.pump2MainActive
	out 4 "статус: по кол-ву включений" <= #127.byCounterActive
	#128 OR(pin 7, startInitializer)
	out 5 "статус: по наработке" <= #127.byWorkTimeActive
	#129 ND0502manager:TwoPumpManager(startStopPump1: #127.startPump1, startStopPump2: #127.startPump2, alarmPump1: #130, alarmPump2: #131, alarmReset: pin 10, counterStart: #127.startByCounter, Pump1ResetCounter: pin 11, Pump2ResetCounter: pin 12, ValueToResetCounter: -, workTimeStart: #127.startByWorkTime, workTimePump1Reset: pin 13, workTimePump2Reset: pin 14)
	out 12 "сигнал на включение насоса 1" <= #129.pump1ON
	#130 NOT(pin 8)
	out 13 "сигнал на включение насоса 2" <= #129.pump2ON
	out 8 "счетчик включений насоса 1" <= #129.counterPump1
	#131 NOT(pin 9)
	out 9 "счетчик включений насоса 2" <= #129.counterPump2
	out 10 "счетчик наработки насоса 1" <= #129.currentWorkTimePump1
	out 11 "счетчик наработки насоса 2" <= #129.currentWorkTimePump2
END_MACRO
#132 ND0502dosingError <= #122.out 1
#133 ND0502statRegimeP1M <= #122.out 2
#134 ND0502statRegimeP2M <= #122.out 3
#135 ND0502statRegimeByC <= #122.out 4
#136 ND0502statRegimeByWT <= #122.out 5
#137 DD1_AO3 <= #122.out 6
#138 DD10_AO0 <= #122.out 7
#139 ND0502counterP1 <= #122.out 8
#140 ND0502counterP2 <= #122.out 9
#141 ND0502workTimeP1 <= #122.out 10
#142 ND0502workTimeP2 <= #122.out 11
#143 DD4_DO.4 <= #122.out 12
#144 DD4_DO.5 <= #122.out 13
#145 AND(DD2_DO.1, DD5_DI.4)
#146 N0105statStartedP1 <= #145
#147 AND(DD5_DI.4, DD2_DO.2)
#148 N0105statStartedP2 <= #147
#149 MACRO Наполнение РЧВ02.03 (заслонка ЗДЭ02.25)(pin 1 "LS02.02раб.верх.уровень РЧВ": DD6_DI.14, pin 2 "LSA02.01 Перелив РЧВ": DD6_DI.13, pin 3 "статус ЗДЭ02.25 открыт": DD9_DI.0, pin 4 "статус ЗДЭ02.25 закрыт": DD9_DI.1, pin 5 "сброс аварий": alarmReset, pin 6 "время на открытие/закрытие": timeToOpenCloseValve)
	#150 OR(testZDE0225, pin 1)
	#151 NOT(pin 1)
	#152 ZDE0225:SimpleValve(inputOpen: #150, inputClose: #153, statusOpen: pin 3, statusClose: pin 4, reset: pin 5, timeToOpenClose: pin 6)
	out 1 "выход на открытие ЗДЭ02.25" <= #152.outputOpen
	#153 OR(#151, #154)
	out 2 "выход на закрытие ЗДЭ02.25" <= #152.outputClose
	out 3 "авария на открытие ЗДЭ02.25" <= #152.errorToOpen
	#154 NOT(pin 2)
	out 4 "авария на закрытие ЗДЭ02.25" <= #152.errorToClose
END_MACRO
#155 DD4_DO.0 <= #149.out 1
#156 DD4_DO.1 <= #149.out 2
#157 ZDE0225errorToOpen <= #149.out 3
#158 ZDE0225errorToClose <= #149.out 4
#159 MACRO управление Н02.04 (подача из РЧВ)(pin 1 "промывка ФС02.01/01": DD6_DI.20, pin 2 "промывка ФС02.01/02": DD6_DI.22, pin 3 "промывка ФС02.01/03": DD6_DI.24, pin 4 "промывка ФС02.01/04": DD6_DI.26, pin 5 "промывка ФС02.01/05": DD6_DI.28, pin 6 "промывка ФС02.01/06": DD6_DI.30, pin 7 "промывка ФС02.02/01": DD7_DI.0, pin 8 "промывка ФС02.02/02": DD7_DI.2, pin 9 "промывка ФС02.02/03": DD7_DI.4, pin 10 "промывка ФС02.02/04": DD7_DI.6, pin 11 "промывка ФС02.02/05": DD7_DI.8, pin 12 "промывка ФС02.02/06": DD7_DI.10, pin 13 "открыт КЭМ05.01": DD1_DI11, pin 14 "открыт КЭМ06.01": DD1_DI10, pin 15 "открыт КЭМ07.01": DD1_DI9, pin 16 "открыт КЭМ08.01": DD1_DI8, pin 17 "сухой ход Н02.04 (0=сух.ход)": DD5_DI.11, pin 18 "выбрать режим: Н02.04/01 - главный": N0204regimeP1M, pin 19 "выбрать режим: Н02.04/02 - главный": N0204regimeP2M, pin 20 "выбрать режим: по кол-ву включений": N0204regimeByC, pin 21 "выбрать режим: по наработке": N0204regimeWT, pin 22 "авария Н02.04/01 (0=авария)": DD5_DI.7, pin 23 "авария Н02.04/02 (0=авария)": DD5_DI.8, pin 24 "сброс аварий": alarmReset, pin 25 "сброс счетчика включений Н02.04/01": N0204resetCountP1, pin 26 "сброс счетчика включений Н02.04/02": N0204resetCountP2, pin 27 "сброс счетчика наработки Н02.04/01": N0204resetWorkTimeP1, pin 28 "сброс счетчика наработки Н02.04/02": N0204resetWorkTimeP2)
	(* Проверка, что фильтры 1 / ступени в регенерации (промывке) *)
	(* Проверка, что фильтры 2 / ступени в регенерации (промывке) *)
	(* Удержание сигнала на выключение насосов для / гарантированного сброса самоподхвата реле. *)
	(* Контроль открытия хотя бы одного из клапанов КЭМ *)
	(* сброс самоподхвата реле *)
	(* Защита от сухого хода Н02.04 / (LS02.03) 0=сух.ход *)
	#160 OR(pin 1, pin 2, pin 3, pin 4, pin 5, pin 6)
	#161 OR(#160, #162, #163)
	#162 OR(pin 7, pin 8, pin 9, pin 10, pin 11, pin 12)
	#163 OR(pin 13, pin 14, pin 15, pin 16)
	#164 N020401fTrigStop:F_TRIG(CLK: #171.pump1ON)
	#165 AND(#161, pin 17)
	#166 OR(#164.Q, #169.Q)
	#167 N0204stop:TOF(IN: #166, PT: T#1s)
	out 5 "стоп Н02.04" <= #167.Q
	#168 N0204chooseRegime:choosePumpRegime(start: #165, pump1Main: pin 18, pump2Main: pin 19, byCounter: #170, byWorkTime: pin 21)
	out 1 "выбран режим Н02.04/01 = главный" <= #168.pump1MainActive
	#169 N020402fTrigStop:F_TRIG(CLK: #171.pump2ON)
	out 2 "выбран режим Н02.04/02 = главный" <= #168.pump2MainActive
	out 3 "выбран режим по кол-ву включений" <= #168.byCounterActive
	#170 OR(pin 20, startInitializer)
	out 4 "выбран режим по наработке" <= #168.byWorkTimeActive
	#171 N0204manager:TwoPumpManager(startStopPump1: #168.startPump1, startStopPump2: #168.startPump2, alarmPump1: NOT pin 22, alarmPump2: NOT pin 23, alarmReset: pin 24, counterStart: #168.startByCounter, Pump1ResetCounter: pin 25, Pump2ResetCounter: pin 26, ValueToResetCounter: -, workTimeStart: #168.startByWorkTime, workTimePump1Reset: pin 27, workTimePump2Reset: pin 28)
	out 6 "пуск Н02.04/01" <= #171.pump1ON
	out 7 "пуск Н02.04/02" <= #171.pump2ON
	out 8 "счетчик включений Н02.04/01" <= #171.counterPump1
	out 9 "счетчик включений Н02.04/02" <= #171.counterPump2
	out 10 "счетчик наработки Н02.04/01" <= #171.currentWorkTimePump1
	out 11 "счетчик наработки Н02.04/02" <= #171.currentWorkTimePump2
END_MACRO
#172 N0204statRegimeP1M <= #159.out 1
#173 N0204statRegimeP2M <= #159.out 2
#174 N0204statRegimeByC <= #159.out 3
#175 N0204statRegimeWT <= #159.out 4
#176 DD4_DO.14 <= #159.out 5
#177 DD1_DO1 <= #159.out 6
#178 DD1_DO2 <= #159.out 7
#179 N0204counterP1 <= #159.out 8
#180 N0204counterP2 <= #159.out 9
#181 N0204workTimeP1 <= #159.out 10
#182 N0204workTimeP2 <= #159.out 11
#183 MACRO управление НД06.02 УПК(pin 1 "вход расходомера в куб/час": DD1_AI2_FT0102value, pin 2 "max производительность НД в мл/мин": ND0602setMaxDosVal, pin 3 "задание дозирования в мл/куб": ND0602setKoefProp, pin 4 "режим:1 насос главный": ND0602regimeP1M, pin 5 "режим: 2 насос главный": ND0602regimeP2M, pin 6 "режим: по наработке": ND0602regimeByWT, pin 7 "режим: по кол-ву включений": ND0602regimeByC, pin 8 "авария 1 насоса": DD6_DI.2, pin 9 "авария 2 насоса": DD6_DI.3, pin 10 "сброс аварий": alarmReset, pin 11 "сброс счетчика включений 1 насоса": ND0602resetCountP1, pin 12 "сброс ссчетчика включений 2 насоса": ND0602resetCountP2, pin 13 "сброс наработки 1 насоса": ND0602resetWorkTimeP1, pin 14 "сброс наработки 2 насоса": ND0602resetWorkTimeP2)
	(* сигнал 4...20мА на НД06.02/02 *)
	(* сигнал 4...20мА на НД06.02/01 *)
	(* Если на входе SEL = TRUE, / то нижнее значение, / иначе - то,что посередине. *)
	#184 SEL(#191.pump1ON, 0, #186.outputValue)
	#185 REAL_TO_WORD(#184)
	out 6 "выход 4...20мА насоса 1" <= #185
	#186 ND0602dosing:DosingPumpProportional(flowValue: pin 1, setMinPumpDosingValue: -, setMaxPumpDosingValue: pin 2, minOutputValue: -, maxOutputValue: -, setKoeffProportionality: pin 3, minFlowToStart: -)
	out 1 "ошибка блока дозирования" <= #186.dosingError
	#187 SEL(#191.pump2ON, 0, #186.outputValue)
	#188 REAL_TO_WORD(#187)
	out 7 "выход 4...20мА насоса 2" <= #188
	#189 ND0602regime:choosePumpRegime(start: #186.startDosingPump, pump1Main: pin 4, pump2Main: pin 5, byCounter: #190, byWorkTime: pin 6)
	out 2 "статус: 1 насос главный" <= #189.pump1MainActive
	out 3 "статус: 2 насос главный" <= #189.pump2MainActive
	out 4 "статус: по кол-ву включений" <= #189.byCounterActive
	#190 OR(pin 7, startInitializer)
	out 5 "статус: по наработке" <= #189.byWorkTimeActive
	#191 ND0602manager:TwoPumpManager(startStopPump1: #189.startPump1, startStopPump2: #189.startPump2, alarmPump1: #192, alarmPump2: #193, alarmReset: pin 10, counterStart: #189.startByCounter, Pump1ResetCounter: pin 11, Pump2ResetCounter: pin 12, ValueToResetCounter: -, workTimeStart: #189.startByWorkTime, workTimePump1Reset: pin 13, workTimePump2Reset: pin 14)
	out 12 "сигнал на включение насоса 1" <= #191.pump1ON
	#192 NOT(pin 8)
	out 13 "сигнал на включение насоса 2" <= #191.pump2ON
	out 8 "счетчик включений насоса 1" <= #191.counterPump1
	#193 NOT(pin 9)
	out 9 "счетчик включений насоса 2" <= #191.counterPump2
	out 10 "счетчик наработки насоса 1" <= #191.currentWorkTimePump1
	out 11 "счетчик наработки насоса 2" <= #191.currentWorkTimePump2
END_MACRO
#194 ND0602dosingError <= #183.out 1
#195 ND0602statRegimeP1M <= #183.out 2
#196 ND0602statRegimeP2M <= #183.out 3
#197 ND0602statRegimeByC <= #183.out 4
#198 ND0602statRegimeByWT <= #183.out 5
#199 DD10_AO1 <= #183.out 6
#200 DD10_AO2 <= #183.out 7
#201 ND0602counterP1 <= #183.out 8
#202 ND0602counterP2 <= #183.out 9
#203 ND0602workTimeP1 <= #183.out 10
#204 ND0602workTimeP2 <= #183.out 11
#205 DD4_DO.6 <= #183.out 12
#206 DD4_DO.7 <= #183.out 13
#207 OR(errorToOpenZDE0301, errorToCloseZDE0301, errorToOpenZDE0302, errorToCloseZDE0302)
#208 OR(DD5_DI.27, #207)
#209 OR(#207, DD5_DI.29)
#210 MACRO Работа УФО03.01(pin 1 "Работа УФО03.01/01": DD5_DI.26, pin 2 "Работа УФО03.01/02": DD5_DI.28, pin 3 "Значение расхода от FT01.02": DD1_AI2_FT0102value, pin 4 "мин.допустимый расход для насосов Н01.05": N0105minFlow, pin 5 "Задержка включения УФО на создание потока": UFO0301startDelayTime, pin 6 "выбор режим: УФО03.01/01 главное": UFO0301regimeP1M, pin 7 "выбор режим: УФО03.01/02 главное": UFO0301regimeP2M, pin 8 "выбор режим: по кол-ву включений": UFO0301regimeByC, pin 9 "выбор режим: по наработке": UFO0301regimeWT, pin 10 "авария УФО03.01/01": #208, pin 11 "авария УФО03.01/02": #209, pin 12 "сброс аварий": alarmReset, pin 13 "сброс счетчика включений УФО03.01/01": UFO0301resetCountP1, pin 14 "сброс счетчика включений УФО03.01/02": UFO0301resetCountP2, pin 15 "сброс счетчика наработки УФО03.01/01": UFO0301resetWorkTimeP1, pin 16 "сброс счетчика наработки УФО03.01/02": UFO0301resetWorkTimeP2)
	(* Контроль, если УФО включили вручную, / а потока при этом нет. *)
	(* Для подачи предостережения на пульте / оператора (при необходимости), а также / сигнализации лампой АВАРИЯ. *)
	(* Задержка старта УФО *)
	(* Включаем УФО, если расходомер показывает расход больше, / чем заданный как минимально допустимый для работы насосов Н01.05. *)
	#211 OR(pin 1, pin 2)
	#212 AND(#211, #213)
	out 1 "УФО вкл без потока" <= #212
	#213 NOT(#215.Q)
	#214 GE(pin 3, pin 4)
	#215 UFO0301startDelay:TON(IN: #214, PT: pin 5)
	#216 UFO0301regimeManager:choosePumpRegime(start: #215.Q, pump1Main: pin 6, pump2Main: pin 7, byCounter: #217, byWorkTime: pin 9)
	out 2 "активен режим - главное УФО 03.01/01" <= #216.pump1MainActive
	out 3 "активен режим - главное УФО 03.01/02" <= #216.pump2MainActive
	out 4 "активен режим - по кол-ву включений" <= #216.byCounterActive
	#217 OR(startInitializer, pin 8)
	out 5 "активен режим - по наработке" <= #216.byWorkTimeActive
	#218 UFO0301manager:TwoPumpManager(startStopPump1: #216.startPump1, startStopPump2: #216.startPump2, alarmPump1: pin 10, alarmPump2: pin 11, alarmReset: pin 12, counterStart: #216.startByCounter, Pump1ResetCounter: pin 13, Pump2ResetCounter: pin 14, ValueToResetCounter: -, workTimeStart: #216.startByWorkTime, workTimePump1Reset: pin 15, workTimePump2Reset: pin 16)
	out 6 "авт. пуск УФО03.01/01" <= #218.pump1ON
	out 7 "авт. пуск УФО03.01/02" <= #218.pump2ON
	out 8 "счетчик включений УФО03.01/01" <= #218.counterPump1
	out 9 "счетчик включений УФО03.01/02" <= #218.counterPump2
	out 10 "счетчик наработки УФО03.01/01" <= #218.currentWorkTimePump1
	out 11 "счетчик наработки УФО03.01/02" <= #218.currentWorkTimePump2
END_MACRO
#219 UFO0301noFlowAttention <= #210.out 1
#220 UFO0301statRegimeP1M <= #210.out 2
#221 UFO0301statRegimeP2M <= #210.out 3
#222 UFO0301statRegimeByC <= #210.out 4
#223 UFO0301statRegimeWT <= #210.out 5
#224 UFO0301counterP1 <= #210.out 8
#225 UFO0301counterP2 <= #210.out 9
#226 UFO0301workTimeP1 <= #210.out 10
#227 UFO0301workTimeP2 <= #210.out 11
#228 MACRO работа задвижек перед УФО и автом.пуск(pin 1 "сигнал на пуск УФО03.01/01": #210.out 6, pin 2 "сигнал на пуск УФО03.01/02": #210.out 7)
	(* авт.пускУФО03.01/02 *)
	(* авт.пускУФО03.01/01 *)
	(* 1 = тест задвижек ЗДЭ / 0 = возможность автом.пуска УФО *)
	(* 1 = открыть ЗДЭ03.01 / 0 = закрыть ЗДЭ03.01 *)
	(* 1 = открыть ЗДЭ03.02 / 0 = закрыть ЗДЭ03.02 *)
	#229 NOT(testZDE03)
	#230 NOT(testZDE03)
	#231 AND(#229, #233, DD1_DI12)
	#232 DD1_DO8 <= #231
	#233 SEL(testZDE03, pin 1, manualZDE0301)
	#234 ZDE0301:SimpleValve(inputOpen: #233, inputClose: NOT #233, statusOpen: DD1_DI12, statusClose: DD1_DI13, reset: alarmReset, timeToOpenClose: timeToOpenCloseValve)
	#235 DD4_DO.16 <= #234.outputOpen
	#236 DD4_DO.17 <= #234.outputClose
	#237 errorToOpenZDE0301 <= #234.errorToOpen
	#238 errorToCloseZDE0301 <= #234.errorToClose
	#239 AND(#230, #241, DD1_DI14)
	#240 DD1_DO9 <= #239
	#241 SEL(testZDE03, pin 2, manualZDE0302)
	#242 ZDE0302:SimpleValve(inputOpen: #241, inputClose: NOT #241, statusOpen: DD1_DI14, statusClose: DD1_DI15, reset: alarmReset, timeToOpenClose: timeToOpenCloseValve)
	#243 DD4_DO.18 <= #242.outputOpen
	#244 DD4_DO.19 <= #242.outputClose
	#245 errorToOpenZDE0302 <= #242.errorToOpen
	#246 errorToCloseZDE0302 <= #242.errorToClose
END_MACRO
#247 MACRO управление НД06.03 УПК(pin 1 "вход расходомера в куб/час": DD1_AI1_FT0101value, pin 2 "max производительность НД в мл/мин": ND0603setMaxDosVal, pin 3 "задание дозирования в мл/куб": ND0603setKoefProp, pin 4 "режим:1 насос главный": ND0603regimeP1M, pin 5 "режим: 2 насос главный": ND0603regimeP2M, pin 6 "режим: по наработке": ND0603regimeByWT, pin 7 "режим: по кол-ву включений": ND0603regimeByC, pin 8 "авария 1 насоса": DD6_DI.4, pin 9 "авария 2 насоса": DD6_DI.5, pin 10 "сброс аварий": alarmReset, pin 11 "сброс счетчика включений 1 насоса": ND0603resetCountP1, pin 12 "сброс ссчетчика включений 2 насоса": ND0603resetCountP2, pin 13 "сброс наработки 1 насоса": ND0603resetWorkTimeP1, pin 14 "сброс наработки 2 насоса": ND0603resetWorkTimeP2)
	(* сигнал 4...20мА на НД06.03/02 *)
	(* сигнал 4...20мА на НД06.03/01 *)
	(* Если на входе SEL = TRUE, / то нижнее значение, / иначе - то,что посередине. *)
	#248 SEL(#255.pump1ON, 0, #250.outputValue)
	#249 REAL_TO_WORD(#248)
	out 6 "выход 4...20мА насоса 1" <= #249
	#250 ND0603dosing:DosingPumpProportional(flowValue: pin 1, setMinPumpDosingValue: -, setMaxPumpDosingValue: pin 2, minOutputValue: -, maxOutputValue: -, setKoeffProportionality: pin 3, minFlowToStart: -)
	out 1 "ошибка блока дозирования" <= #250.dosingError
	#251 SEL(#255.pump2ON, 0, #250.outputValue)
	#252 REAL_TO_WORD(#251)
	out 7 "выход 4...20мА насоса 2" <= #252
	#253 ND0603regime:choosePumpRegime(start: #250.startDosingPump, pump1Main: pin 4, pump2Main: pin 5, byCounter: #254, byWorkTime: pin 6)
	out 2 "статус: 1 насос главный" <= #253.pump1MainActive
	out 3 "статус: 2 насос главный" <= #253.pump2MainActive
	out 4 "статус: по кол-ву включений" <= #253.byCounterActive
	#254 OR(pin 7, startInitializer)
	out 5 "статус: по наработке" <= #253.byWorkTimeActive
	#255 ND0603manager:TwoPumpManager(startStopPump1: #253.startPump1, startStopPump2: #253.startPump2, alarmPump1: #256, alarmPump2: #257, alarmReset: pin 10, counterStart: #253.startByCounter, Pump1ResetCounter: pin 11, Pump2ResetCounter: pin 12, ValueToResetCounter: -, workTimeStart: #253.startByWorkTime, workTimePump1Reset: pin 13, workTimePump2Reset: pin 14)
	out 12 "сигнал на включение насоса 1" <= #255.pump1ON
	#256 NOT(pin 8)
	out 13 "сигнал на включение насоса 2" <= #255.pump2ON
	out 8 "счетчик включений насоса 1" <= #255.counterPump1
	#257 NOT(pin 9)
	out 9 "счетчик включений насоса 2" <= #255.counterPump2
	out 10 "счетчик наработки насоса 1" <= #255.currentWorkTimePump1
	out 11 "счетчик наработки насоса 2" <= #255.currentWorkTimePump2
END_MACRO
#258 ND0603dosingError <= #247.out 1
#259 ND0603statRegimeP1M <= #247.out 2
#260 ND0603statRegimeP2M <= #247.out 3
#261 ND0603statRegimeByC <= #247.out 4
#262 ND0603statRegimeByWT <= #247.out 5
#263 DD10_AO3 <= #247.out 6
#264 DD10_AO4 <= #247.out 7
#265 ND0603counterP1 <= #247.out 8
#266 ND0603counterP2 <= #247.out 9
#267 ND0603workTimeP1 <= #247.out 10
#268 ND0603workTimeP2 <= #247.out 11
#269 DD4_DO.8 <= #247.out 12
#270 DD4_DO.9 <= #247.out 13
#271 MACRO управление Н04.04 (дренажные)(pin 1 "защита от сухого хода Н04.04": DD5_DI.18, pin 2 "автоматич.пускН04.04": DD5_DI.19, pin 3 "режим Н04.04/01 главный": N0404regimeP1M, pin 4 "режим Н04.04/02 главный": N0404regimeP2M, pin 5 "режим по кол-ву включений": N0404regimeByC, pin 6 "режим по наработке": N0404regimeWT, pin 7 "авария Н04.04/01": DD5_DI.15, pin 8 "авария Н04.04/02": DD5_DI.14, pin 9 "сброс аварий": alarmReset, pin 10 "сброс счетчика включений Н04.04/01": N0404resetCountP1, pin 11 "сброс счетчика включений Н04.04/02": N0404resetCountP2, pin 12 "сброс счетчика наработки Н04.04/01": N0404resetWorkTimeP1, pin 13 "сброс счетчика наработки Н04.04/02": N0404resetWorkTimeP2)
	(* сбрасывает самоподхват пускового реле *)
	(* Излишняя перестраховка по сухому ходу, / на уровне реле уже все отрабатывается. *)
	(* насосы имеют электрическую блокировку / от одновременного включения *)
	(* от поплавка *)
	(* сухой ход Н04.04 / 0=защита *)
	(* 0=авария *)
	#272 NOT(pin 1)
	out 1 "стоп Н04.04" <= #272
	#273 AND(pin 1, pin 2)
	#274 N0401choosePumpRegime:choosePumpRegime(start: #273, pump1Main: pin 3, pump2Main: pin 4, byCounter: #275, byWorkTime: pin 6)
	out 2 "выбран режим: Н04.04/01 главный" <= #274.pump1MainActive
	out 3 "выбран режим: Н04.04/02 главный" <= #274.pump2MainActive
	out 4 "выбран режим: по кол-ву включений" <= #274.byCounterActive
	#275 OR(startInitializer, pin 5)
	out 5 "выбран режим: по наработке" <= #274.byWorkTimeActive
	#276 N0404twoPumpManager:TwoPumpManager(startStopPump1: #274.startPump1, startStopPump2: #274.startPump2, alarmPump1: #277, alarmPump2: #278, alarmReset: pin 9, counterStart: #274.startByCounter, Pump1ResetCounter: pin 10, Pump2ResetCounter: pin 11, ValueToResetCounter: -, workTimeStart: #274.startByWorkTime, workTimePump1Reset: pin 12, workTimePump2Reset: pin 13)
	out 6 "пуск Н04.04/01" <= #276.pump1ON
	#277 NOT(pin 7)
	out 7 "пуск Н04.04/02" <= #276.pump2ON
	out 8 "счетчик кол-ва включений Н04.04/01" <= #276.counterPump1
	#278 NOT(pin 8)
	out 9 "счетчик кол-ва включений Н04.04/02" <= #276.counterPump2
	out 10 "счетчик времени наработки Н04.04/01" <= #276.currentWorkTimePump1
	out 11 "счетчик времени наработки Н04.04/02" <= #276.currentWorkTimePump2
END_MACRO
#279 DD4_DO.15 <= #271.out 1
#280 N0404statRegimeP1M <= #271.out 2
#281 N0404statRegimeP2M <= #271.out 3
#282 N0404statRegimeByC <= #271.out 4
#283 N0404statRegimeWT <= #271.out 5
#284 DD1_DO5 <= #271.out 6
#285 DD1_DO6 <= #271.out 7
#286 N0404counterP1 <= #271.out 8
#287 N0404counterP2 <= #271.out 9
#288 N0404workTimeP1 <= #271.out 10
#289 N0404workTimeP2 <= #271.out 11
#290 MACRO управление НД07.03 УПЩ (поддержка рН, ПИД-регулятор)(pin 1 "вход рН-метра QE01.01": DD1_AI3_QE0101value, pin 2 "уставка рН": ND0703pHsetValue, pin 3 "режим:1 насос главный": ND0703regimeP1M, pin 4 "режим: 2 насос главный": ND0703regimeP2M, pin 5 "режим: по наработке": ND0703regimeByWT, pin 6 "режим: по кол-ву включений": ND0703regimeByC, pin 7 "авария 1 насоса": DD6_DI.6, pin 8 "авария 2 насоса": DD6_DI.7, pin 9 "сброс аварий": alarmReset, pin 10 "сброс счетчика включений 1 насоса": ND0703resetCountP1, pin 11 "сброс счетчика включений 2 насоса": ND0703resetCountP2, pin 12 "сброс наработки 1 насоса": ND0703resetWorkTimeP1, pin 13 "сброс наработки 2 насоса": ND0703resetWorkTimeP2, pin 14 "ручное управл.выходом Y (4...20мА)": ND0703YoutManual, pin 15 "1=ручное/0=автомат.управл.": ND0703YmanAuto, pin 16 "вход расходомера FT01.01 (куб.м/час)": DD1_AI1_FT0101value, pin 17 "коэфф.I": ND0703koeffI, pin 18 "коэфф.D": ND0703koeffD, pin 19 "коэфф.Р": ND0703koeffP)
	(* сигнал 4...20мА на НД07.03/02 *)
	(* сигнал 4...20мА на НД07.03/01 *)
	(* Если на входе SEL = TRUE, / то нижнее значение, / иначе - то,что посередине. *)
	(* min расход в кубометрах в час / для неачала дозирования. *)
	#291 ND0703pidReg:PID(ACTUAL: pin 1, SET_POINT: pin 2, KP: pin 19, TN: pin 17, TV: pin 18, Y_MANUAL: pin 14, Y_OFFSET: 12, Y_MIN: 4, Y_MAX: 20, MANUAL: pin 15, RESET: #291.OVERFLOW)
	#292 SEL(#299.pump1ON, 0, #291.Y)
	#293 REAL_TO_WORD(#292)
	out 5 "выход 4...20мА насоса 1" <= #293
	#294 SEL(#299.pump2ON, 0, #291.Y)
	#295 REAL_TO_WORD(#294)
	out 6 "выход 4...20мА насоса 2" <= #295
	#296 GE(pin 16, 10)
	#297 ND0703regime:choosePumpRegime(start: #296, pump1Main: pin 3, pump2Main: pin 4, byCounter: #298, byWorkTime: pin 5)
	out 1 "статус: 1 насос главный" <= #297.pump1MainActive
	out 2 "статус: 2 насос главный" <= #297.pump2MainActive
	out 3 "статус: по кол-ву включений" <= #297.byCounterActive
	out 4 "статус: по наработке" <= #297.byWorkTimeActive
	#298 OR(pin 6, startInitializer)
	#299 ND0703manager:TwoPumpManager(startStopPump1: #297.startPump1, startStopPump2: #297.startPump2, alarmPump1: #300, alarmPump2: #301, alarmReset: pin 9, counterStart: #297.startByCounter, Pump1ResetCounter: pin 10, Pump2ResetCounter: pin 11, ValueToResetCounter: -, workTimeStart: #297.startByWorkTime, workTimePump1Reset: pin 12, workTimePump2Reset: pin 13)
	out 11 "сигнал на включение насоса 1" <= #299.pump1ON
	#300 NOT(pin 7)
	out 12 "сигнал на включение насоса 2" <= #299.pump2ON
	out 7 "счетчик включений насоса 1" <= #299.counterPump1
	#301 NOT(pin 8)
	out 8 "счетчик включений насоса 2" <= #299.counterPump2
	out 9 "счетчик наработки насоса 1" <= #299.currentWorkTimePump1
	out 10 "счетчик наработки насоса 2" <= #299.currentWorkTimePump2
END_MACRO
#302 ND0703statRegimeP1M <= #290.out 1
#303 ND0703statRegimeP2M <= #290.out 2
#304 ND0703statRegimeByC <= #290.out 3
#305 ND0703statRegimeByWT <= #290.out 4
#306 DD10_AO5 <= #290.out 5
#307 DD10_AO6 <= #290.out 6
#308 ND0703counterP1 <= #290.out 7
#309 ND0703counterP2 <= #290.out 8
#310 ND0703workTimeP1 <= #290.out 9
#311 ND0703workTimeP2 <= #290.out 10
#312 DD4_DO.10 <= #290.out 11
#313 DD4_DO.11 <= #290.out 12
#314 MACRO импульсный счетчик FQS0301(pin 1 "вход от счетчика": DD6_DI.19, pin 2 "вес импульса счетчика": FQS0301impulsValue, pin 3 "сброс счетчика": FQS0301reset, pin 4 "величина коррекции счетчика": FQS0301correction, pin 5 "прибавить коррекцию": FQS0301addCorrection, pin 6 "вычесть коррекцию": FQS0301deleteCorrection)
	(* сброс показаний счетчика *)
	(* значение в REAL (в какой-то момент начинает / отображаться в экспоненциальной форме) *)
	(* Если в результате коррекции накопленная сумма станет меньше нуля, то она принудительно станет равна нулю. *)
	(* коррекция показаний счетчика. *)
	(* число, коорое будем прибавлять или / вычитать из накопленной суммы стоков. *)
	#315 FQS0301rTrig:R_TRIG(CLK: pin 1)
	#316 ADD(EN: #315.Q, FQS0301totalAmount, pin 2)
	out 1 "накопленная сумма стоков (REAL)" <= #316
	#317 FQS0301resetRtrig:R_TRIG(CLK: pin 3)
	#318 MOVE(EN: #317.Q, 0)
	#319 FQS0301totalAmount <= #318
	#320 FQS0301addCorrRtrig:R_TRIG(CLK: pin 5)
	#321 ADD(EN: #320.Q, FQS0301totalAmount, pin 4)
	#322 FQS0301totalAmount <= #321
	#323 FQS0301deleteCorrRtrig:R_TRIG(CLK: pin 6)
	#324 SUB(EN: #323.Q, FQS0301totalAmount, pin 4)
	#325 FQS0301totalAmount <= #324
	#326 LT(FQS0301totalAmount, 0)
	#327 MOVE(EN: #326, 0)
	#328 FQS0301totalAmount <= #327
END_MACRO
#329 FQS0301totalAmount <= #314.out 1
#330 MACRO управление НД08.03 УПФ(pin 1 "вход расходомера в куб/час": DD1_AI1_FT0101value, pin 2 "max производительность НД в мл/мин": ND0803setMaxDosVal, pin 3 "задание дозирования в мл/куб": ND0803setKoefProp, pin 4 "режим:1 насос главный": ND0803regimeP1M, pin 5 "режим: 2 насос главный": ND0803regimeP2M, pin 6 "режим: по наработке": ND0803regimeByWT, pin 7 "режим: по кол-ву включений": ND0803regimeByC, pin 8 "авария 1 насоса": DD5_DI.12, pin 9 "авария 2 насоса": DD5_DI.13, pin 10 "сброс аварий": alarmReset, pin 11 "сброс счетчика включений 1 насоса": ND0803resetCountP1, pin 12 "сброс ссчетчика включений 2 насоса": ND0803resetCountP2, pin 13 "сброс наработки 1 насоса": ND0803resetWorkTimeP1, pin 14 "сброс наработки 2 насоса": ND0803resetWorkTimeP2, pin 15 "сухой ход 1 насоса": DD1_DI6, pin 16 "сухой ход 2 насоса": DD1_DI7)
	(* сигнал 4...20мА на НД08.03/02 *)
	(* сигнал 4...20мА на НД08.03/01 *)
	(* Если на входе SEL = TRUE, / то нижнее значение, / иначе - то,что посередине. *)
	#331 SEL(#340.pump1ON, 0, #332.outputValue)
	out 6 "выход 4...20мА насоса 1" <= #331
	#332 ND0803dosing:DosingPumpProportional(flowValue: pin 1, setMinPumpDosingValue: -, setMaxPumpDosingValue: pin 2, minOutputValue: -, maxOutputValue: -, setKoeffProportionality: pin 3, minFlowToStart: -)
	out 1 "ошибка блока дозирования" <= #332.dosingError
	#333 SEL(#340.pump2ON, 0, #332.outputValue)
	out 7 "выход 4...20мА насоса 2" <= #333
	#334 ND0803regime:choosePumpRegime(start: #332.startDosingPump, pump1Main: pin 4, pump2Main: pin 5, byCounter: #335, byWorkTime: pin 6)
	out 2 "статус: 1 насос главный" <= #334.pump1MainActive
	out 3 "статус: 2 насос главный" <= #334.pump2MainActive
	out 4 "статус: по кол-ву включений" <= #334.byCounterActive
	#335 OR(pin 7, startInitializer)
	out 5 "статус: по наработке" <= #334.byWorkTimeActive
	out 12 "сигнал на включение насоса 1" <= #340.pump1ON
	#336 NOT(pin 8)
	#337 OR(#336, pin 15)
	out 13 "сигнал на включение насоса 2" <= #340.pump2ON
	#338 NOT(pin 9)
	#339 OR(#338, pin 16)
	#340 ND0803manager:TwoPumpManager(startStopPump1: #334.startPump1, startStopPump2: #334.startPump2, alarmPump1: #337, alarmPump2: #339, alarmReset: pin 10, counterStart: #334.startByCounter, Pump1ResetCounter: pin 11, Pump2ResetCounter: pin 12, ValueToResetCounter: -, workTimeStart: #334.startByWorkTime, workTimePump1Reset: pin 13, workTimePump2Reset: pin 14)
	out 8 "счетчик включений насоса 1" <= #340.counterPump1
	out 9 "счетчик включений насоса 2" <= #340.counterPump2
	out 10 "счетчик наработки насоса 1" <= #340.currentWorkTimePump1
	out 11 "счетчик наработки насоса 2" <= #340.currentWorkTimePump2
END_MACRO
#341 ND0803dosingError <= #330.out 1
#342 ND0803statRegimeP1M <= #330.out 2
#343 ND0803statRegimeP2M <= #330.out 3
#344 ND0803statRegimeByC <= #330.out 4
#345 ND0803statRegimeByWT <= #330.out 5
#346 DD1_AO1 <= #330.out 6
#347 DD1_AO2 <= #330.out 7
#348 ND0803counterP1 <= #330.out 8
#349 ND0803counterP2 <= #330.out 9
#350 ND0803workTimeP1 <= #330.out 10
#351 ND0803workTimeP2 <= #330.out 11
#352 DD1_DO3 <= #330.out 12
#353 DD1_DO4 <= #330.out 13
#354 AND(DD1_DI5, DD1_DI4, DD6_DI.11)
#355 DD1_DO8 <= #354
#356 EQ(lastError, 0)
#357 alarmPLKnetworkDelay:TOF(IN: #356, PT: T#20s)
#358 NOT(#357.Q)
#359 alarmPLKnetwork <= #358
#360 MACRO управление НД08.04 УПФ(pin 1 "насос Н04.01 работает": DD7_DI.13, pin 2 "авария НД08.04": DD6_DI.16, pin 3 "уставкаНД08.04(0...100%)": ND0804doseValue)
	(* Преобразует сигнал 0...100 / пропорционально в 4...20мА *)
	#361 AND(pin 1, pin 2)
	out 1 "пуск/стоп НД08.04" <= #361
	#362 ND0804linearTransformator:LIN_TRAFO(IN: pin 3, IN_MIN: 0, IN_MAX: 100, OUT_MIN: 4, OUT_MAX: 20)
	#363 REAL_TO_WORD(#362.OUT)
	out 2 "управление НД08.04 (4...20мА)" <= #363
	out 3 "ошибка блока дозирования" <= #362.ERROR
END_MACRO
#364 DD4_DO.12 <= #360.out 1
#365 DD10_AO7 <= #360.out 2
#366 ND0804dosingError <= #360.out 3
#367 NOT(DD6_DI.0)
#368 alarmND050201 <= #367
#369 NOT(DD6_DI.23)
#370 alarmFS020102 <= #369
#371 NOT(DD9_DI.14)
#372 alarmZDE0211power <= #371
#373 NOT(DD6_DI.1)
#374 alarmND050202 <= #373
#375 NOT(DD6_DI.25)
#376 alarmFS020103 <= #375
#377 NOT(DD9_DI.15)
#378 alarmZDE0212power <= #377
#379 NOT(DD6_DI.2)
#380 alarmND060201 <= #379
#381 NOT(DD6_DI.27)
#382 alarmFS020104 <= #381
#383 NOT(DD9_DI.16)
#384 alarmZDE0213power <= #383
#385 NOT(DD6_DI.3)
#386 alarmND060202 <= #385
#387 NOT(DD6_DI.29)
#388 alarmFS020105 <= #387
#389 NOT(DD9_DI.17)
#390 alarmZDE0214power <= #389
#391 MACRO контроль включения мешалок(pin 1 "работа НД06.02/01": DD4_DO.6, pin 2 "работа НД06.02/02": DD4_DO.7, pin 3 "работа НД06.03/01": DD4_DO.8, pin 4 "работа НД06.03/02": DD4_DO.9, pin 5 "работа мешалки М06.04": DD5_DI.21, pin 6 "работа НД07.03/01": DD4_DO.10, pin 7 "работа НД07.03/02": DD4_DO.11, pin 8 "работа мешалки М07.02": DD5_DI.23, pin 9 "работа НД08.03/01": DD1_DO3, pin 10 "работа НД08.03/02": DD1_DO4, pin 11 "работа НД08.04": DD4_DO.12, pin 12 "работа мешалки М08.02": DD5_DI.25)
	#392 OR(pin 1, pin 2, pin 3, pin 4)
	#393 AND(#392, #394)
	out 1 "дозирования при выключенной М06.04" <= #393
	#394 NOT(pin 5)
	#395 OR(pin 6, pin 7)
	#396 AND(#395, #397)
	out 2 "дозирования при выключенной М07.02" <= #396
	#397 NOT(pin 8)
	#398 OR(pin 9, pin 10, pin 11)
	#399 AND(#398, #400)
	out 3 "дозирования при выключенной М08.02" <= #399
	#400 NOT(pin 12)
END_MACRO
#401 M0604attention <= #391.out 1
#402 M0702attention <= #391.out 2
#403 M0802attention <= #391.out 3
#404 NOT(DD6_DI.4)
#405 alarmND060301 <= #404
#406 NOT(DD6_DI.31)
#407 alarmFS020106 <= #406
#408 NOT(DD9_DI.18)
#409 alarmZDE0215power <= #408
#410 NOT(DD6_DI.5)
#411 alarmND060302 <= #410
#412 NOT(DD7_DI.1)
#413 alarmFS020201 <= #412
#414 NOT(DD9_DI.19)
#415 alarmZDE0216power <= #414
#416 NOT(DD6_DI.6)
#417 alarmND070301 <= #416
#418 NOT(DD7_DI.3)
#419 alarmFS020202 <= #418
#420 NOT(DD9_DI.20)
#421 alarmZDE0217power <= #420
#422 NOT(DD6_DI.7)
#423 alarmND070302 <= #422
#424 NOT(DD7_DI.5)
#425 alarmFS020203 <= #424
#426 NOT(DD9_DI.21)
#427 alarmZDE0218power <= #426
#428 NOT(DD5_DI.12)
#429 alarmND080301 <= #428
#430 NOT(DD7_DI.7)
#431 alarmFS020204 <= #430
#432 NOT(DD9_DI.22)
#433 alarmZDE0219power <= #432
#434 NOT(DD5_DI.13)
#435 alarmND080302 <= #434
#436 NOT(DD7_DI.9)
#437 alarmFS020205 <= #436
#438 NOT(DD9_DI.23)
#439 alarmZDE0220power <= #438
#440 NOT(DD6_DI.16)
#441 alarmND0804 <= #440
#442 NOT(DD7_DI.11)
#443 alarmFS020206 <= #442
#444 NOT(DD9_DI.24)
#445 alarmZDE0221power <= #444
#446 NOT(DD6_DI.11)
#447 alarmOGM0104overload <= #446
#448 NOT(DD9_DI.4)
#449 alarmZDE0201power <= #448
#450 NOT(DD9_DI.25)
#451 alarmZDE0222power <= #450
#452 MACRO переменные для обмена с панелью()
	#453 MACRO PSW регистры на передачу в панель (отображение)()
		(* PSW регистры на передачу в панель (отображение) *)
		(* panFQS0301totalAmount - переменная отображена сразу на выходе соответствующего макроса (учет очищенных стоков). / Здесь не хранится. *)
		#454 panFT0101value <= DD1_AI1_FT0101value
		#455 panQE0101value <= DD1_AI3_QE0101value
		#456 panFT0102value <= DD1_AI2_FT0102value
		#457 panQE0102value <= DD1_AI4_QE0102value
		#458 panFPKpressureValue <= DD1_AI5_FPKpressureValue
		#459 panFQS0301total <= FQS0301totalAmount
		#460 panTemperature <= temperatureValue
		#461 MACRO Время наработки и кол-во включений агрегатов()
			#462 workTimeND050201:TimeFromWorkTime(input: ND0502workTimeP1)
			#463 panND050201workDays <= #462.days
			#464 panND050201workHours <= #462.hours
			#465 panND050201workMinutes <= #462.minutes
			#466 panND050201workSeconds <= #462.seconds
			#467 workTimeND050202:TimeFromWorkTime(input: ND0502workTimeP2)
			#468 panND050202workDays <= #467.days
			#469 panND050202workHours <= #467.hours
			#470 panND050202workMinutes <= #467.minutes
			#471 panND050202workSeconds <= #467.seconds
			#472 panND0502counterP1 <= ND0502counterP1
			#473 panND0502counterP2 <= ND0502counterP2
			#474 workTimeND060201:TimeFromWorkTime(input: ND0602workTimeP1)
			#475 panND060201workDays <= #474.days
			#476 panND060201workHours <= #474.hours
			#477 panND060201workMinutes <= #474.minutes
			#478 panND060201workSeconds <= #474.seconds
			#479 workTimeND060202:TimeFromWorkTime(input: ND0602workTimeP2)
			#480 panND060202workDays <= #479.days
			#481 panND060202workHours <= #479.hours
			#482 panND060202workMinutes <= #479.minutes
			#483 panND060202workSeconds <= #479.seconds
			#484 panND0602counterP1 <= ND0602counterP1
			#485 panND0602counterP2 <= ND0602counterP2
			#486 workTimeND060301:TimeFromWorkTime(input: ND0603workTimeP1)
			#487 panND060301workDays <= #486.days
			#488 panND060301workHours <= #486.hours
			#489 panND060301workMinutes <= #486.minutes
			#490 panND060301workSeconds <= #486.seconds
			#491 workTimeND060302:TimeFromWorkTime(input: ND0603workTimeP2)
			#492 panND060302workDays <= #491.days
			#493 panND060302workHours <= #491.hours
			#494 panND060302workMinutes <= #491.minutes
			#495 panND060302workSeconds <= #491.seconds
			#496 panND0603counterP1 <= ND0603counterP1
			#497 panND0603counterP2 <= ND0603counterP2
			#498 workTimeND070301:TimeFromWorkTime(input: ND0703workTimeP1)
			#499 panND070301workDays <= #498.days
			#500 panND070301workHours <= #498.hours
			#501 panND070301workMinutes <= #498.minutes
			#502 panND070301workSeconds <= #498.seconds
			#503 workTimeND070302:TimeFromWorkTime(input: ND0703workTimeP2)
			#504 panND070302workDays <= #503.days
			#505 panND070302workHours <= #503.hours
			#506 panND070302workMinutes <= #503.minutes
			#507 panND070302workSeconds <= #503.seconds
			#508 panND0703counterP1 <= ND0703counterP1
			#509 panND0703counterP2 <= ND0703counterP2
			#510 workTimeND080301:TimeFromWorkTime(input: ND0803workTimeP1)
			#511 panND080301workDays <= #510.days
			#512 panND080301workHours <= #510.hours
			#513 panND080301workMinutes <= #510.minutes
			#514 panND080301workSeconds <= #510.seconds
			#515 workTimeND080302:TimeFromWorkTime(input: ND0803workTimeP2)
			#516 panND080302workDays <= #515.days
			#517 panND080302workHours <= #515.hours
			#518 panND080302workMinutes <= #515.minutes
			#519 panND080302workSeconds <= #515.seconds
			#520 panND0803counterP1 <= ND0803counterP1
			#521 panND0803counterP2 <= ND0803counterP2
			#522 workTimeN010501:TimeFromWorkTime(input: N0105workTimeP1)
			#523 panN010501workDays <= #522.days
			#524 panN010501workHours <= #522.hours
			#525 panN010501workMinutes <= #522.minutes
			#526 panN010501workSeconds <= #522.seconds
			#527 workTimeN010502:TimeFromWorkTime(input: N0105workTimeP2)
			#528 panN010502workDays <= #527.days
			#529 panN010502workHours <= #527.hours
			#530 panN010502workMinutes <= #527.minutes
			#531 panN010502workSeconds <= #527.seconds
			#532 panN0105counterP1 <= N0105counterP1
			#533 panN0105counterP2 <= N0105counterP2
			#534 workTimeN020401:TimeFromWorkTime(input: N0204workTimeP1)
			#535 panN020401workDays <= #534.days
			#536 panN020401workHours <= #534.hours
			#537 panN020401workMinutes <= #534.minutes
			#538 panN020401workSeconds <= #534.seconds
			#539 workTimeN020402:TimeFromWorkTime(input: N0204workTimeP2)
			#540 panN020402workDays <= #539.days
			#541 panN020402workHours <= #539.hours
			#542 panN020402workMinutes <= #539.minutes
			#543 panN020402workSeconds <= #539.seconds
			#544 panN0204counterP1 <= N0204counterP1
			#545 panN0204counterP2 <= N0204counterP2
			#546 workTimeN040401:TimeFromWorkTime(input: N0404workTimeP1)
			#547 panN040401workDays <= #546.days
			#548 panN040401workHours <= #546.hours
			#549 panN040401workMinutes <= #546.minutes
			#550 panN040401workSeconds <= #546.seconds
			#551 workTimeN040402:TimeFromWorkTime(input: N0404workTimeP2)
			#552 panN040402workDays <= #551.days
			#553 panN040402workHours <= #551.hours
			#554 panN040402workMinutes <= #551.minutes
			#555 panN040402workSeconds <= #551.seconds
			#556 panN0404counterP1 <= N0404counterP1
			#557 panN0404counterP2 <= N0404counterP2
			#558 workTimeUFO030101:TimeFromWorkTime(input: UFO0301workTimeP1)
			#559 panUFO030101workDays <= #558.days
			#560 panUFO030101workHours <= #558.hours
			#561 panUFO030101workMinutes <= #558.minutes
			#562 panUFO030101workSeconds <= #558.seconds
			#563 workTimeUFO030102:TimeFromWorkTime(input: UFO0301workTimeP2)
			#564 panUFO030102workDays <= #563.days
			#565 panUFO030102workHours <= #563.hours
			#566 panUFO030102workMinutes <= #563.minutes
			#567 panUFO030102workSeconds <= #563.seconds
			#568 panUFO0301counterP1 <= UFO0301counterP1
			#569 panUFO0301counterP2 <= UFO0301counterP2
		END_MACRO
	END_MACRO
	#570 MACRO PSB регистры на передачу в панель (отображение)()
		(* PSB регистры на передачу в панель (отображение) *)
		#571 MACRO 8 bit output module 1()
			#572 panStartND050201 <= DD4_DO.4
			#573 panStartND050202 <= DD4_DO.5
			#574 panStartND060201 <= DD4_DO.6
			#575 panStartND060202 <= DD4_DO.7
			#576 panStartND060301 <= DD4_DO.8
			#577 panStartND060302 <= DD4_DO.9
			#578 panStartM0604 <= DD5_DI.21
			#579 panStartND070301 <= DD4_DO.10
		END_MACRO
		#580 MACRO 8 bit output module 2()
			#581 panStartND070302 <= DD4_DO.11
			#582 panStartM0702 <= DD5_DI.23
			#583 panStartND080301 <= DD1_DO3
			#584 panStartND080302 <= DD1_DO4
			#585 panStartND0804 <= DD4_DO.12
			#586 panStartM0802 <= DD5_DI.25
			#587 panStartN020401 <= DD5_DI.9
			#588 panStartN020402 <= DD5_DI.10
		END_MACRO
		#589 MACRO 8 bit output module 3()
			#590 panStartN010501 <= N0105statStartedP1
			#591 panStartN010502 <= N0105statStartedP2
			#592 panCleanFS020101 <= DD6_DI.20
			#593 panCleanFS020102 <= DD6_DI.22
			#594 panCleanFS020103 <= DD6_DI.24
			#595 panCleanFS020104 <= DD6_DI.26
			#596 panCleanFS020105 <= DD6_DI.28
			#597 panCleanFS020106 <= DD6_DI.30
		END_MACRO
		#598 MACRO 8 bit output module 4()
			#599 panCleanFS020201 <= DD7_DI. 0
			#600 panCleanFS020202 <= DD7_DI. 2
			#601 panCleanFS020203 <= DD7_DI. 4
			#602 panCleanFS020204 <= DD7_DI. 6
			#603 panCleanFS020205 <= DD7_DI. 8
			#604 panCleanFS020206 <= DD7_DI. 10
			#605 panSludgeReady <= DD7_DI.15
			#606 panStartN0401 <= DD7_DI.13
		END_MACRO
		#607 MACRO 8 bit output module 5()
			#608 panKSHE0401open <= DD9_DI.2
			#609 panFPKready <= DD7_DI.12
			#610 panFPKneedToClean <= FPKneedToClean
			#611 panStartN040401 <= DD5_DI.16
			#612 panStartN040402 <= DD5_DI.17
			#613 panStartUFO030101 <= DD5_DI.26
			#614 panStartUFO030102 <= DD5_DI.28
			#615 panAlarm <= alarm
		END_MACRO
		#616 MACRO 8 bit output module 6()
			#617 panErrorTempSensor <= DD1_AI0_error
			#618 panErrorFT0101 <= DD1_AI1_error
			#619 panErrorFT0102 <= DD1_AI2_error
			#620 panErrorQE0102 <= DD1_AI3_error
			#621 panErrorQE0102 <= DD1_AI4_error
			#622 panAlarmHighTemp <= alarmHighTemperature
			#623 panAlarmLowTemp <= alarmLowTemperature
			#624 panND0502dosingError <= ND0502dosingError
		END_MACRO
		#625 MACRO 8 bit output module 7()
			#626 panND0602dosingError <= ND0602dosingError
			#627 panND0603dosingError <= ND0603dosingError
			#628 panND0803dosingError <= ND0803dosingError
			#629 panND0804dosingError <= ND0804dosingError
			#630 panND080301emptyAlarm <= DD1_DI6
			#631 panND080302emptyAlarm <= DD1_DI7
			#632 panN010501alarm <= N010501alarm
			#633 panN010502alarm <= N010502alarm
		END_MACRO
		#634 MACRO 8 bit output module 8()
			#635 panZDE0225errorToOpen <= ZDE0225errorToOpen
			#636 panZDE0225errorToClose <= ZDE0225errorToClose
			#637 panFPKalarm <= DD7_DI.14
			#638 panFPKnotStarted <= FPKnotStarted
			#639 panErrorFPKsensor <= DD1_AI5_error
			#640 panFPKkshe0401errorToOpen <= FPKkshe0401errorToOpen
			#641 panFPKkshe0401errorToClose <= FPKkshe0401errorToClose
			#642 panUFO030101alarm <= DD5_DI.27
		END_MACRO
		#643 MACRO 8 bit output module 9()
			#644 panUFO030102alarm <= DD5_DI.29
			#645 panFilterFailToRegen020101 <= filterFailToRegen020101
			#646 panErrorToOpenZD0201 <= errorToOpenZD0201
			#647 panErrorToCloseZD0201 <= errorToCloseZD0201
			#648 panErrorToOpenZD0207 <= errorToOpenZD0207
			#649 panErrorToCloseZD0207 <= errorToCloseZD0207
			#650 panFilterFailToRegen020102 <= filterFailToRegen020102
			#651 panErrorToOpenZD0202 <= errorToOpenZD0202
		END_MACRO
		#652 MACRO 8 bit output module 10()
			#653 panErrorToCloseZD0202 <= errorToCloseZD0202
			#654 panErrorToOpenZD0208 <= errorToOpenZD0208
			#655 panErrorToCloseZD0208 <= errorToCloseZD0208
			#656 panFilterFailToRegen020103 <= filterFailToRegen020103
			#657 panErrorToOpenZD0203 <= errorToOpenZD0203
			#658 panErrorToCloseZD0203 <= errorToCloseZD0203
			#659 panErrorToOpenZD0209 <= errorToOpenZD0209
			#660 panErrorToCloseZD0209 <= errorToCloseZD0209
		END_MACRO
		#661 MACRO 8 bit output module 11()
			#662 panFilterFailToRegen020104 <= filterFailToRegen020104
			#663 panErrorToOpenZD0204 <= errorToOpenZD0204
			#664 panErrorToCloseZD0204 <= errorToCloseZD0204
			#665 panErrorToOpenZD0210 <= errorToOpenZD0210
			#666 panErrorToCloseZD0210 <= errorToCloseZD0210
			#667 panFilterFailToRegen020105 <= filterFailToRegen020105
			#668 panErrorToOpenZD0205 <= errorToOpenZD0205
			#669 panErrorToCloseZD0205 <= errorToCloseZD0205
		END_MACRO
		#670 MACRO 8 bit output module 12()
			#671 panErrorToOpenZD0211 <= errorToOpenZD0211
			#672 panErrorToCloseZD0211 <= errorToCloseZD0211
			#673 panFilterFailToRegen020106 <= filterFailToRegen020106
			#674 panErrorToOpenZD0206 <= errorToOpenZD0206
			#675 panErrorToCloseZD0206 <= errorToCloseZD0206
			#676 panErrorToOpenZD0212 <= errorToOpenZD0212
			#677 panErrorToCloseZD0212 <= errorToCloseZD0212
			#678 panFilterFailToRegen020201 <= filterFailToRegen020201
		END_MACRO
		#679 MACRO 8 bit output module 13()
			#680 panErrorToOpenZD0213 <= errorToOpenZD0213
			#681 panErrorToCloseZD0213 <= errorToCloseZD0213
			#682 panErrorToOpenZD0219 <= errorToOpenZD0219
			#683 panErrorToCloseZD0219 <= errorToCloseZD0219
			#684 panFilterFailToRegen020202 <= filterFailToRegen020202
			#685 panErrorToOpenZD0214 <= errorToOpenZD0214
			#686 panErrorToCloseZD0214 <= errorToCloseZD0214
			#687 panErrorToOpenZD0220 <= errorToOpenZD0220
		END_MACRO
		#688 MACRO 8 bit output module 14()
			#689 panErrorToCloseZD0220 <= errorToCloseZD0220
			#690 panFilterFailToRegen020203 <= filterFailToRegen020203
			#691 panErrorToOpenZD0215 <= errorToOpenZD0215
			#692 panErrorToCloseZD0215 <= errorToCloseZD0215
			#693 panErrorToOpenZD0221 <= errorToOpenZD0221
			#694 panErrorToCloseZD0221 <= errorToCloseZD0221
			#695 panFilterFailToRegen020204 <= filterFailToRegen020204
			#696 panErrorToOpenZD0216 <= errorToOpenZD0216
		END_MACRO
		#697 MACRO 8 bit output module 15()
			#698 panErrorToCloseZD0216 <= errorToCloseZD0216
			#699 panErrorToOpenZD0222 <= errorToOpenZD0222
			#700 panErrorToCloseZD0222 <= errorToCloseZD0222
			#701 panFilterFailToRegen020205 <= filterFailToRegen020205
			#702 panErrorToOpenZD0217 <= errorToOpenZD0217
			#703 panErrorToCloseZD0217 <= errorToCloseZD0217
			#704 panErrorToOpenZD0223 <= errorToOpenZD0223
			#705 panErrorToCloseZD0223 <= errorToCloseZD0223
		END_MACRO
		#706 MACRO 8 bit output module 16()
			#707 panFilterFailToRegen020206 <= filterFailToRegen020206
			#708 panErrorToOpenZD0218 <= errorToOpenZD0218
			#709 panErrorToCloseZD0218 <= errorToCloseZD0218
			#710 panErrorToOpenZD0224 <= errorToOpenZD0224
			#711 panErrorToCloseZD0224 <= errorToCloseZD0224
			#712 panAlarmPLKnetwork <= alarmPLKnetwork
			#713 panAlarmND050201 <= alarmND050201
			#714 panAlarmND050202 <= alarmND050202
		END_MACRO
		#715 MACRO 8 bit output module 17()
			#716 panAlarmND060201 <= alarmND060201
			#717 panAlarmND060202 <= alarmND060202
			#718 panAlarmND060301 <= alarmND060301
			#719 panAlarmND060302 <= alarmND060302
			#720 panAlarmND070301 <= alarmND070301
			#721 panAlarmND070302 <= alarmND070302
			#722 panAlarmND080301 <= alarmND080301
			#723 panAlarmND080302 <= alarmND080302
		END_MACRO
		#724 MACRO 8 bit output module 18()
			#725 panAlarmND0804 <= alarmND0804
			#726 panAlarmOGM0104overload <= alarmOGM0104overload
			#727 panAlarmRCHV0203overload <= alarmRCHV0203overload
			#728 panAlarmN040402 <= alarmN040402
			#729 panAlarmN040401 <= alarmN040401
			#730 panAlarmM0604 <= alarmM0604
			#731 panAlarmM0702 <= alarmM0702
			#732 panAlarmM0802 <= alarmM0802
		END_MACRO
		#733 MACRO 8 bit output module 19()
			#734 panAlarmN020401 <= alarmN020401
			#735 panAlarmN020402 <= alarmN020402
			#736 panAlarmFS020101 <= alarmFS020101
			#737 panAlarmFS020102 <= alarmFS020102
			#738 panAlarmFS020103 <= alarmFS020103
			#739 panAlarmFS020104 <= alarmFS020104
			#740 panAlarmFS020105 <= alarmFS020105
			#741 panAlarmFS020106 <= alarmFS020106
		END_MACRO
		#742 MACRO 8 bit output module 20()
			#743 panAlarmFS020201 <= alarmFS020201
			#744 panAlarmFS020202 <= alarmFS020202
			#745 panAlarmFS020203 <= alarmFS020203
			#746 panAlarmFS020204 <= alarmFS020204
			#747 panAlarmFS020205 <= alarmFS020205
			#748 panAlarmFS020206 <= alarmFS020206
			#749 panAlarmZDE0201power <= alarmZDE0201power
			#750 panAlarmZDE0202power <= alarmZDE0202power
		END_MACRO
		#751 MACRO 8 bit output module 21()
			#752 panAlarmZDE0203power <= alarmZDE0203power
			#753 panAlarmZDE0204power <= alarmZDE0204power
			#754 panAlarmZDE0205power <= alarmZDE0205power
			#755 panAlarmZDE0206power <= alarmZDE0206power
			#756 panAlarmZDE0207power <= alarmZDE0207power
			#757 panAlarmZDE0208power <= alarmZDE0208power
			#758 panAlarmZDE0209power <= alarmZDE0209power
			#759 panAlarmZDE0210power <= alarmZDE0210power
		END_MACRO
		#760 MACRO 8 bit output module 22()
			#761 panAlarmZDE0211power <= alarmZDE0211power
			#762 panAlarmZDE0212power <= alarmZDE0212power
			#763 panAlarmZDE0213power <= alarmZDE0213power
			#764 panAlarmZDE0214power <= alarmZDE0214power
			#765 panAlarmZDE0215power <= alarmZDE0215power
			#766 panAlarmZDE0216power <= alarmZDE0216power
			#767 panAlarmZDE0217power <= alarmZDE0217power
			#768 panAlarmZDE0218power <= alarmZDE0218power
		END_MACRO
		#769 MACRO 8 bit output module 23()
			#770 panAlarmZDE0219power <= alarmZDE0219power
			#771 panAlarmZDE0220power <= alarmZDE0220power
			#772 panAlarmZDE0221power <= alarmZDE0221power
			#773 panAlarmZDE0222power <= alarmZDE0222power
			#774 panAlarmZDE0223power <= alarmZDE0223power
			#775 panAlarmZDE0224power <= alarmZDE0224power
			#776 panAlarmZDE0225power <= alarmZDE0225power
			#777 panAlarmKSHE0401power <= alarmKSHE0401power
		END_MACRO
		#778 MACRO 8 bit output module 24()
			#779 panAlarmKNS <= alarmKNS
			#780 panAlarmPowerSocketFS <= alarmPowerSocketFS
			#781 panAlarmKEMvalvesPower <= alarmKEMvalvesPower
			#782 panAlarmEmergencyPressed <= alarmEmergencyPressed
			#783 panAlarmRKF <= alarmRKF
			#784 panUFO0301noFlowAttention <= UFO0301noFlowAttention
			#785 panM0604attention <= M0604attention
			#786 panM0702attention <= M0702attention
		END_MACRO
		#787 MACRO 8 bit output module 25()
			#788 panM0802attention <= M0802attention
			#789 panStatusKNS <= DD6_DI.8
			#790 panND0502statRegimeP1M <= ND0502statRegimeP1M
			#791 panND0502statRegimeP2M <= ND0502statRegimeP2M
			#792 panND0502statRegimeByC <= ND0502statRegimeByC
			#793 panND0502statRegimeByWT <= ND0502statRegimeByWT
			#794 panND0602statRegimeP1M <= ND0602statRegimeP1M
			#795 panND0602statRegimeP2M <= ND0602statRegimeP2M
		END_MACRO
		#796 MACRO 8 bit output module 26()
			#797 panND0602statRegimeByC <= ND0602statRegimeByC
			#798 panND0602statRegimeByWT <= ND0602statRegimeByWT
			#799 panND0603statRegimeP1M <= ND0603statRegimeP1M
			#800 panND0603statRegimeP2M <= ND0603statRegimeP2M
			#801 panND0603statRegimeByC <= ND0603statRegimeByC
			#802 panND0603statRegimeByWT <= ND0603statRegimeByWT
			#803 panND0703statRegimeP1M <= ND0703statRegimeP1M
			#804 panND0703statRegimeP2M <= ND0703statRegimeP2M
		END_MACRO
		#805 MACRO 8 bit output module 27()
			#806 panND0703statRegimeByC <= ND0703statRegimeByC
			#807 panND0703statRegimeByWT <= ND0703statRegimeByWT
			#808 panND0803statRegimeP1M <= ND0803statRegimeP1M
			#809 panND0803statRegimeP2M <= ND0803statRegimeP2M
			#810 panND0803statRegimeByC <= ND0803statRegimeByC
			#811 panND0803statRegimeByWT <= ND0803statRegimeByWT
			#812 panN0105statRegimeP1M <= N0105statRegimeP1M
			#813 panN0105statRegimeP2M <= N0105statRegimeP2M
		END_MACRO
		#814 MACRO 8 bit output module 28()
			#815 panN0105statRegimeByC <= N0105statRegimeByC
			#816 panN0105statRegimeByWT <= N0105statRegimeByWT
			#817 panN0204statRegimeP1M <= N0204statRegimeP1M
			#818 panN0204statRegimeP2M <= N0204statRegimeP2M
			#819 panN0204statRegimeByC <= N0204statRegimeByC
			#820 panN0204statRegimeWT <= N0204statRegimeWT
			#821 panN0404statRegimeP1M <= N0404statRegimeP1M
			#822 panN0404statRegimeP2M <= N0404statRegimeP2M
		END_MACRO
		#823 MACRO 8 bit output module 29()
			#824 panN0404statRegimeByC <= N0404statRegimeByC
			#825 panN0404statRegimeWT <= N0404statRegimeWT
			#826 panUFO0301statRegimeP1M <= UFO0301statRegimeP1M
			#827 panUFO0301statRegimeP2M <= UFO0301statRegimeP2M
			#828 panUFO0301statRegimeByC <= UFO0301statRegimeByC
			#829 panUFO0301statRegimeWT <= UFO0301statRegimeWT
			#830 panZDE0225open <= DD9_DI.0
			#831 panZDE0201open <= DD7_DI.16
		END_MACRO
		#832 MACRO 8 bit output module 30()
			#833 panZDE0201close <= DD7_DI.17
			#834 panZDE0202open <= DD7_DI.18
			#835 panZDE0202close <= DD7_DI.19
			#836 panZDE0203open <= DD7_DI.20
			#837 panZDE0203close <= DD7_DI.21
			#838 panZDE0204open <= DD7_DI.22
			#839 panZDE0204close <= DD7_DI.23
			#840 panZDE0205open <= DD7_DI.24
		END_MACRO
		#841 MACRO 8 bit output module 31()
			#842 panZDE0205close <= DD7_DI.25
			#843 panZDE0206open <= DD7_DI.26
			#844 panZDE0206close <= DD7_DI.27
			#845 panZDE0207open <= DD7_DI.28
			#846 panZDE0207close <= DD7_DI.29
			#847 panZDE0208open <= DD7_DI.30
			#848 panZDE0208close <= DD7_DI.31
			#849 panZDE0209open <= DD8_DI.0
		END_MACRO
		#850 MACRO 8 bit output module 32()
			#851 panZDE0209close <= DD8_DI.1
			#852 panZDE0210open <= DD8_DI.2
			#853 panZDE0210close <= DD8_DI.3
			#854 panZDE0211open <= DD8_DI.4
			#855 panZDE0211close <= DD8_DI.5
			#856 panZDE0212open <= DD8_DI.6
			#857 panZDE0212close <= DD8_DI.7
			#858 panZDE0213open <= DD8_DI.8
		END_MACRO
		#859 MACRO 8 bit output module 33()
			#860 panZDE0213close <= DD8_DI.9
			#861 panZDE0214open <= DD8_DI.10
			#862 panZDE0214close <= DD8_DI.11
			#863 panZDE0215open <= DD8_DI.12
			#864 panZDE0215close <= DD8_DI.13
			#865 panZDE0216open <= DD8_DI.14
			#866 panZDE0216close <= DD8_DI.15
			#867 panZDE0217open <= DD8_DI.16
		END_MACRO
		#868 MACRO 8 bit output module 34()
			#869 panZDE0217close <= DD8_DI.17
			#870 panZDE0218open <= DD8_DI.18
			#871 panZDE0218close <= DD8_DI.19
			#872 panZDE0219open <= DD8_DI.20
			#873 panZDE0219close <= DD8_DI.21
			#874 panZDE0220open <= DD8_DI.22
			#875 panZDE0220close <= DD8_DI.23
			#876 panZDE0221open <= DD8_DI.24
		END_MACRO
		#877 MACRO 8 bit output module 35()
			#878 panZDE0221close <= DD8_DI.25
			#879 panZDE0222open <= DD8_DI.26
			#880 panZDE0222close <= DD8_DI.27
			#881 panZDE0223open <= DD8_DI.28
			#882 panZDE0223close <= DD8_DI.29
			#883 panZDE0224open <= DD8_DI.30
			#884 panZDE0224close <= DD8_DI.31
			#885 panZDE0225close <= DD9_DI.1
		END_MACRO
		#886 MACRO 8 bit output module 36x()
			#887 panKSHE0401close <= DD9_DI.3
			#888 panZDE0301open <= DD1_DI12
			#889 panZDE0301close <= DD1_DI13
			#890 panZDE0302open <= DD1_DI14
			#891 panZDE0302close <= DD1_DI15
			#892 panErrorToOpenZDE0301 <= errorToOpenZDE0301
			#893 panErrorToCloseZDE0301 <= errorToCloseZDE0301
			#894 panErrorToOpenZDE0302 <= errorToOpenZDE0302
		END_MACRO
		#895 panErrorToCloseZDE0302 <= errorToCloseZDE0302
		#896 panAlarmZDE0301power <= alarmZDE0301power
		#897 panAlarmZDE0302power <= alarmZDE0302power
	END_MACRO
	#898 MACRO PFW регистры на чтение из панели (управление ПЛК)()
		#899 MUL(panTimeToOpenCloseValve, 1000)
		#900 REAL_TO_TIME(#899)
		#901 TimeToOpenCloseValve <= #900
		#902 maxTemperature <= panMaxTemperature
		#903 minTemperature <= panMinTemperature
		#904 ND0502setMaxDosVal <= panND0502setMaxDosVal
		#905 ND0502setKoefProp <= panND0502setKoefProp
		#906 ND0602setMaxDosVal <= panND0602setMaxDosVal
		#907 ND0602setKoefProp <= panND0602setKoefProp
		#908 ND0603setMaxDosVal <= panND0603setMaxDosVal
		#909 ND0603setKoefProp <= panND0603setKoefProp
		#910 ND0703pHsetValue <= panND0703pHsetValue
		#911 ND0703YoutManual <= panND0703YoutManual
		#912 ND0703koeffI <= panND0703koeffI
		#913 ND0703koeffD <= panND0703koeffD
		#914 ND0703koeffP <= panND0703koeffP
		#915 ND0803setMaxDosVal <= panND0803setMaxDosVal
		#916 ND0803setKoefProp <= panND0803setKoefProp
		#917 ND0804doseValue <= panND0804doseValue
		#918 N0105flowSetValue <= panN0105flowSetValue
		#919 N0105YoutManual <= panN0105YoutManual
		#920 N0105koeffI <= panN0105koeffI
		#921 N0105koeffD <= panN0105koeffD
		#922 N0105koeffP <= panN0105koeffP
		#923 FQS0301impulsValue <= panFQS0301impulsValue
		#924 FQS0301correction <= panFQS0301correction
		#925 MUL(panFPKtimeToWork, 1000)
		#926 REAL_TO_TIME(#925)
		#927 FPKtimeToWork <= #926
		#928 MUL(panFPKnotStartedTime, 1000)
		#929 REAL_TO_TIME(#928)
		#930 FPKnotStartedTime <= #929
		#931 FPKmaxPressureValue <= panFPKmaxPressureValue
		#932 filterValueToRegen <= panFilterValueToRegen
	END_MACRO
	#933 MACRO PSB регистры на чтение из панели (управление ПЛК)()
		(* PSB регистры на чтение из панели (управление ПЛК) *)
		#934 MACRO 8 bit input module 1()
			#935 alarmReset <= panAlarmResetButton
			#936 ND0502resetCountP1 <= panND0502resetCountP1
			#937 ND0502resetCountP2 <= panND0502resetCountP2
			#938 ND0502resetWorkTimeP1 <= panND0502resetWorkTimeP1
			#939 ND0502resetWorkTimeP2 <= panND0502resetWorkTimeP2
			#940 ND0502regimeP1M <= panND0502regimeP1M
			#941 ND0502regimeP2M <= panND0502regimeP2M
			#942 ND0502regimeByC <= panND0502regimeByC
		END_MACRO
		#943 MACRO 8 bit input module 2()
			#944 ND0502regimeByWT <= panND0502regimeByWT
			#945 ND0602resetCountP1 <= panND0602resetCountP1
			#946 ND0602resetCountP2 <= panND0602resetCountP2
			#947 ND0602resetWorkTimeP1 <= panND0602resetWorkTimeP1
			#948 ND0602resetWorkTimeP2 <= panND0602resetWorkTimeP2
			#949 ND0602regimeP1M <= panND0602regimeP1M
			#950 ND0602regimeP2M <= panND0602regimeP2M
			#951 ND0602regimeByC <= panND0602regimeByC
		END_MACRO
		#952 MACRO 8 bit input module 3()
			#953 ND0602regimeByWT <= panND0602regimeByWT
			#954 ND0603resetCountP1 <= panND0603resetCountP1
			#955 ND0603resetCountP2 <= panND0603resetCountP2
			#956 ND0603resetWorkTimeP1 <= panND0603resetWorkTimeP1
			#957 ND0603resetWorkTimeP2 <= panND0603resetWorkTimeP2
			#958 ND0603regimeP1M <= panND0603regimeP1M
			#959 ND0603regimeP2M <= panND0603regimeP2M
			#960 ND0603regimeByC <= panND0603regimeByC
		END_MACRO
		#961 MACRO 8 bit input module 4()
			#962 ND0603regimeByWT <= panND0603regimeByWT
			#963 ND0703resetCountP1 <= panND0703resetCountP1
			#964 ND0703resetCountP2 <= panND0703resetCountP2
			#965 ND0703resetWorkTimeP1 <= panND0703resetWorkTimeP1
			#966 ND0703resetWorkTimeP2 <= panND0703resetWorkTimeP2
			#967 ND0703regimeP1M <= panND0703regimeP1M
			#968 ND0703regimeP2M <= panND0703regimeP2M
			#969 ND0703regimeByC <= panND0703regimeByC
		END_MACRO
		#970 MACRO 8 bit input module 5()
			#971 ND0703regimeByWT <= panND0703regimeByWT
			#972 ND0703YmanAuto <= panND0703YmanAuto
			#973 ND0803resetCountP1 <= panND0803resetCountP1
			#974 ND0803resetCountP2 <= panND0803resetCountP2
			#975 ND0803resetWorkTimeP1 <= panND0803resetWorkTimeP1
			#976 ND0803resetWorkTimeP2 <= panND0803resetWorkTimeP2
			#977 ND0803regimeP1M <= panND0803regimeP1M
			#978 ND0803regimeP2M <= panND0803regimeP2M
		END_MACRO
		#979 MACRO 8 bit input module 6()
			#980 ND0803regimeByC <= panND0803regimeByC
			#981 ND0803regimeByWT <= panND0803regimeByWT
			#982 N0105resetCountP1 <= panN0105resetCountP1
			#983 N0105resetCountP2 <= panN0105resetCountP2
			#984 N0105resetWorkTimeP1 <= panN0105resetWorkTimeP1
			#985 N0105resetWorkTimeP2 <= panN0105resetWorkTimeP2
			#986 N0105regimeByC <= panN0105regimeByC
			#987 N0105regimeByWT <= panN0105regimeByWT
		END_MACRO
		#988 MACRO 8 bit input module 7()
			#989 N0105YmanAuto <= panN0105YmanAuto
			#990 N0204resetCountP1 <= panN0204resetCountP1
			#991 N0204resetCountP2 <= panN0204resetCountP2
			#992 N0204resetWorkTimeP1 <= panN0204resetWorkTimeP1
			#993 N0204resetWorkTimeP2 <= panN0204resetWorkTimeP2
			#994 N0204regimeP1M <= panN0204regimeP1M
			#995 N0204regimeP2M <= panN0204regimeP2M
			#996 N0204regimeByC <= panN0204regimeByC
		END_MACRO
		#997 MACRO 8 bit input module 8()
			#998 N0204regimeWT <= panN0204regimeWT
			#999 UFO0301resetCountP1 <= panUFO0301resetCountP1
			#1000 UFO0301resetCountP2 <= panUFO0301resetCountP2
			#1001 UFO0301resetWorkTimeP1 <= panUFO0301resetWorkTimeP1
			#1002 UFO0301resetWorkTimeP2 <= panUFO0301resetWorkTimeP2
			#1003 UFO0301regimeP1M <= panUFO0301regimeP1M
			#1004 UFO0301regimeP2M <= panUFO0301regimeP2M
			#1005 UFO0301regimeByC <= panUFO0301regimeByC
		END_MACRO
		#1006 MACRO 8 bit input module 9()
			#1007 UFO0301regimeWT <= panUFO0301regimeWT
			#1008 N0404resetCountP1 <= panN0404resetCountP1
			#1009 N0404resetCountP2 <= panN0404resetCountP2
			#1010 N0404resetWorkTimeP1 <= panN0404resetWorkTimeP1
			#1011 N0404resetWorkTimeP2 <= panN0404resetWorkTimeP2
			#1012 N0404regimeP1M <= panN0404regimeP1M
			#1013 N0404regimeP2M <= panN0404regimeP2M
			#1014 N0404regimeByC <= panN0404regimeByC
		END_MACRO
		#1015 MACRO 8 bit input module 10-11()
			(* одули 10 и 11 заполнены переменными для тестирования задвижек. / Здесь они не показаны, т.к. спешка. / Они вставлены напрямую в макросы управления промывкой фильтров. / testValvesFS020101 - testValvesFS020206 (PSB612-623) *)
			#1016 N0404regimeWT <= panN0404regimeWT
			#1017 FQS0301reset <= panFQS0301reset
			#1018 FQS0301addCorrection <= panFQS0301addCorrection
			#1019 FQS0301deleteCorrection <= panFQS0301deleteCorrection
		END_MACRO
		#1020 testKSHE0401 <= panTestKSHE0401
		#1021 testZDE0225 <= panTestZDE0225
		#1022 testZDE03 <= panTestZDE03
		#1023 manualZDE0301 <= panManualZDE0301
		#1024 manualZDE0302 <= panManualZDE0302
	END_MACRO
END_MACRO
#1025 NOT(DD6_DI.13)
#1026 alarmRCHV0203overload <= #1025
#1027 NOT(DD9_DI.5)
#1028 alarmZDE0202power <= #1027
#1029 NOT(DD9_DI.26)
#1030 alarmZDE0223power <= #1029
#1031 MACRO переменные на диспетчеризацию()
	#1032 remFT0101value <= DD1_AI1_FT0101value
	#1033 remFQS0301totalAmount <= FQS0301totalAmount
	#1034 remTemperatureValue <= temperatureValue
	#1035 remStatusN010501started <= N0105statStartedP1
	#1036 remStatusN010502started <= N0105statStartedP2
	#1037 remStatusUFO030101started <= DD5_DI.26
	#1038 remStatusUFO030102started <= DD5_DI.28
	#1039 remAlarm <= Alarm
	#1040 remN010501alarm <= N010501alarm
	#1041 remN010502alarm <= N010502alarm
	#1042 remFPKalarm <= DD7_DI.14
	#1043 remUFO030101alarm <= DD5_DI.27
	#1044 remUFO030102alarm <= DD5_DI.29
	#1045 remAlarmEmergencyPressed <= alarmEmergencyPressed
	#1046 remAlarmOOGM0104overload <= DD6_DI.11
	#1047 remAlarmRCHV0203overload <= DD6_DI.13
END_MACRO
#1048 NOT(DD5_DI.14)
#1049 alarmN040402 <= #1048
#1050 NOT(DD9_DI.6)
#1051 alarmZDE0203power <= #1050
#1052 NOT(DD9_DI.27)
#1053 alarmZDE0224power <= #1052
#1054 NOT(DD5_DI.15)
#1055 alarmN040401 <= #1054
#1056 NOT(DD9_DI.7)
#1057 alarmZDE0204power <= #1056
#1058 NOT(DD9_DI.28)
#1059 alarmZDE0225power <= #1058
#1060 NOT(DD5_DI.20)
#1061 alarmM0604 <= #1060
#1062 NOT(DD9_DI.8)
#1063 alarmZDE0205power <= #1062
#1064 NOT(DD9_DI.29)
#1065 alarmKSHE0401power <= #1064
#1066 NOT(DD5_DI.22)
#1067 alarmM0702 <= #1066
#1068 NOT(DD9_DI.9)
#1069 alarmZDE0206power <= #1068
#1070 NOT(DD6_DI.9)
#1071 alarmKNS <= #1070
#1072 NOT(DD5_DI.24)
#1073 alarmM0802 <= #1072
#1074 NOT(DD9_DI.10)
#1075 alarmZDE0207power <= #1074
#1076 NOT(DD6_DI.17)
#1077 alarmPowerSocketFS <= #1076
#1078 NOT(DD5_DI.7)
#1079 alarmN020401 <= #1078
#1080 NOT(DD9_DI.11)
#1081 alarmZDE0208power <= #1080
#1082 NOT(DD6_DI.18)
#1083 alarmKEMvalvesPower <= #1082
#1084 NOT(DD5_DI.8)
#1085 alarmN020402 <= #1084
#1086 NOT(DD9_DI.12)
#1087 alarmZDE0209power <= #1086
#1088 NOT(DD1_DI4)
#1089 alarmEmergencyPressed <= #1088
#1090 GT(DD1_AI2_FT0102value, 0)
#1091 filterPulserGen:PulsePerSec(start: #1090)
#1092 DIV(DD1_AI2_FT0102value, 3600)
#1093 ADD(EN: #1091.out, #1092, filterTotalAmountFT0102)
#1094 filterTotalAmountFT0102 <= #1093
#1095 NOT(DD6_DI.21)
#1096 alarmFS020101 <= #1095
#1097 NOT(DD9_DI.13)
#1098 alarmZDE0210power <= #1097
#1099 NOT(DD1_DI5)
#1100 alarmRKF <= #1099
#1101 NOT(DD9_DI.30)
#1102 alarmZDE0301power <= #1101
#1103 NOT(DD9_DI.31)
#1104 alarmZDE0302power <= #1103
#1105 MOVE(EN: filterTotalAmountReset, 0)
#1106 filterTotalAmountFT0102 <= #1105
#1107 GE(filterTotalAmountFT0102, filterValueToRegen)
#1108 MACRO управление промывкой фильтра ФС02.01.01(pin 1 "сигнал на промывку": #1107, pin 2 "авария фильтра": DD6_DI.21, pin 3 "подтверждение промывки": DD6_DI.20, pin 4 "сброс аварий": alarmReset, pin 5 "начать очередь снова": filterStartNewQueue, pin 6 "ЗДЭ02.01 открыта": DD7_DI.16, pin 7 "ЗДЭ02.01 закрыта": DD7_DI.17, pin 8 "ЗДЭ02.07 открыта": DD7_DI.28, pin 9 "ЗДЭ02.07 закрыта": DD7_DI.29, pin 10 "время движения ЗДЭ": timeToOpenCloseValve, pin 11 "авария питания ЗДЭ02.01": DD9_DI.4, pin 12 "авария питания ЗДЭ02.07": DD9_DI.10)
	(* <- выход использовать в / последнем фильтре для / начала очереди заново *)
	(* если открыт = промывка *)
	(* если открыт = фильтрация *)
	out 1 "следующий в очереди" <= #1111.output
	out 2 "промыть ФС02.01.01" <= #1110
	#1109 ZD0201:SimpleValve(inputOpen: NOT #1110, inputClose: #1110, statusOpen: pin 6, statusClose: pin 7, reset: pin 4, timeToOpenClose: pin 10)
	out 6 "открыть ЗДЭ02.01" <= #1109.outputOpen
	out 7 "закрыть ЗДЭ02.01" <= #1109.outputClose
	out 8 "авария открытия ЗДЭ02.01" <= #1109.errorToOpen
	#1110 OR(panTestValvesFS020101, #1111.regenFilterOUT)
	out 9 "авария закрытия ЗДЭ02.01" <= #1109.errorToClose
	#1111 FS020101manager:FilterQueueManager(input: pin 1, filterAlarm: #1112, regenFilterStatus: pin 3, alarmReset: pin 4, startNextLoop: pin 5)
	#1112 OR(alarmZD020107, pin 2, pin 11, pin 12)
	out 3 "ФС02.01.01 промыт" <= #1111.regenerated
	out 4 "не удалось промыть" <= #1111.failToRegen
	#1113 OR(#1109.errorToOpen, #1109.errorToClose, #1115.errorToOpen, #1115.errorToClose)
	#1114 alarmZD020107 <= #1113
	out 5 "сброс счетчика" <= #1111.counterReset
	#1115 ZD0207:SimpleValve(inputOpen: #1110, inputClose: NOT #1110, statusOpen: pin 8, statusClose: pin 9, reset: pin 4, timeToOpenClose: pin 10)
	out 10 "открыть ЗДЭ02.07" <= #1115.outputOpen
	out 11 "закрыть ЗДЭ02.07" <= #1115.outputClose
	out 12 "авария открытия ЗДЭ02.07" <= #1115.errorToOpen
	out 13 "авария закрытия ЗДЭ02.07" <= #1115.errorToClose
END_MACRO
#1116 DD2_DO.4 <= #1108.out 2
#1117 regeneratedFS020101 <= #1108.out 3
#1118 filterFailToRegen020101 <= #1108.out 4
#1119 filterTotalAmountReset <= #1108.out 5
#1120 DD2_DO.16 <= #1108.out 6
#1121 DD2_DO.17 <= #1108.out 7
#1122 errorToOpenZD0201 <= #1108.out 8
#1123 errorToCloseZD0201 <= #1108.out 9
#1124 DD2_DO.28 <= #1108.out 10
#1125 DD2_DO.29 <= #1108.out 11
#1126 errorToOpenZD0207 <= #1108.out 12
#1127 errorToCloseZD0207 <= #1108.out 13
#1128 MACRO управление промывкой фильтра ФС02.01.02(pin 1 "сигнал на промывку": #1108.out 1, pin 2 "авария фильтра": DD6_DI.23, pin 3 "подтверждение промывки": DD6_DI.22, pin 4 "сброс аварий": alarmReset, pin 5 "начать очередь снова": filterStartNewQueue, pin 6 "ЗДЭ02.02 открыта": DD7_DI.18, pin 7 "ЗДЭ02.02 закрыта": DD7_DI.19, pin 8 "ЗДЭ02.08 открыта": DD7_DI.30, pin 9 "ЗДЭ02.08 закрыта": DD7_DI.31, pin 10 "время движения ЗДЭ": timeToOpenCloseValve, pin 11 "авария питания ЗДЭ02.02": DD9_DI.5, pin 12 "авария питания ЗДЭ02.08": DD9_DI.11)
	(* <- выход использовать в / последнем фильтре для / начала очереди заново *)
	(* если открыт = промывка *)
	(* если открыт = фильтрация *)
	out 1 "следующий в очереди" <= #1131.output
	out 2 "промыть ФС02.01.02" <= #1130
	#1129 ZD0202:SimpleValve(inputOpen: NOT #1130, inputClose: #1130, statusOpen: pin 6, statusClose: pin 7, reset: pin 4, timeToOpenClose: pin 10)
	out 5 "открыть ЗДЭ02.02" <= #1129.outputOpen
	out 6 "закрыть ЗДЭ02.02" <= #1129.outputClose
	out 7 "авария открытия ЗДЭ02.02" <= #1129.errorToOpen
	#1130 OR(panTestValvesFS020102, #1131.regenFilterOUT)
	out 8 "авария закрытия ЗДЭ02.02" <= #1129.errorToClose
	#1131 FS020102manager:FilterQueueManager(input: pin 1, filterAlarm: #1132, regenFilterStatus: pin 3, alarmReset: pin 4, startNextLoop: pin 5)
	#1132 OR(alarmZD020208, pin 2, pin 11, pin 12)
	#1133 OR(#1129.errorToOpen, #1129.errorToClose, #1135.errorToOpen, #1135.errorToClose)
	#1134 alarmZD020208 <= #1133
	out 3 "ФС02.01.02 промыт" <= #1131.regenerated
	out 4 "не удалось промыть" <= #1131.failToRegen
	#1135 ZD0208:SimpleValve(inputOpen: #1130, inputClose: NOT #1130, statusOpen: pin 8, statusClose: pin 9, reset: pin 4, timeToOpenClose: pin 10)
	out 9 "открыть ЗДЭ02.08" <= #1135.outputOpen
	out 10 "закрыть ЗДЭ02.08" <= #1135.outputClose
	out 11 "авария открытия ЗДЭ02.08" <= #1135.errorToOpen
	out 12 "авария закрытия ЗДЭ02.08" <= #1135.errorToClose
END_MACRO
#1136 DD2_DO.5 <= #1128.out 2
#1137 regeneratedFS020102 <= #1128.out 3
#1138 filterFailToRegen020102 <= #1128.out 4
#1139 DD2_DO.18 <= #1128.out 5
#1140 DD2_DO.19 <= #1128.out 6
#1141 errorToOpenZD0202 <= #1128.out 7
#1142 errorToCloseZD0202 <= #1128.out 8
#1143 DD2_DO.30 <= #1128.out 9
#1144 DD2_DO.31 <= #1128.out 10
#1145 errorToOpenZD0208 <= #1128.out 11
#1146 errorToCloseZD0208 <= #1128.out 12
#1147 MACRO управление промывкой фильтра ФС02.01.03(pin 1 "сигнал на промывку": #1128.out 1, pin 2 "авария фильтра": DD6_DI.25, pin 3 "подтверждение промывки": DD6_DI.24, pin 4 "сброс аварий": alarmReset, pin 5 "начать очередь снова": filterStartNewQueue, pin 6 "ЗДЭ02.03 открыта": DD7_DI.20, pin 7 "ЗДЭ02.03 закрыта": DD7_DI.21, pin 8 "ЗДЭ02.09 открыта": DD8_DI.0, pin 9 "ЗДЭ02.09 закрыта": DD8_DI.1, pin 10 "время движения ЗДЭ": timeToOpenCloseValve, pin 11 "авария питания ЗДЭ02.03": DD9_DI.6, pin 12 "авария питания ЗДЭ02.09": DD9_DI.12)
	(* <- выход использовать в / последнем фильтре для / начала очереди заново *)
	(* если открыт = промывка *)
	(* если открыт = фильтрация *)
	out 1 "следующий в очереди" <= #1150.output
	out 2 "промыть ФС02.01.03" <= #1149
	#1148 ZD0203:SimpleValve(inputOpen: NOT #1149, inputClose: #1149, statusOpen: pin 6, statusClose: pin 7, reset: pin 4, timeToOpenClose: pin 10)
	out 5 "открыть ЗДЭ02.03" <= #1148.outputOpen
	out 6 "закрыть ЗДЭ02.03" <= #1148.outputClose
	out 7 "авария открытия ЗДЭ02.03" <= #1148.errorToOpen
	#1149 OR(panTestValvesFS020103, #1150.regenFilterOUT)
	out 8 "авария закрытия ЗДЭ02.03" <= #1148.errorToClose
	#1150 FS020103manager:FilterQueueManager(input: pin 1, filterAlarm: #1151, regenFilterStatus: pin 3, alarmReset: pin 4, startNextLoop: pin 5)
	#1151 OR(alarmZD020309, pin 2, pin 11, pin 12)
	#1152 OR(#1148.errorToOpen, #1148.errorToClose, #1154.errorToOpen, #1154.errorToClose)
	#1153 alarmZD020309 <= #1152
	out 3 "ФС02.01.03 промыт" <= #1150.regenerated
	out 4 "не удалось промыть" <= #1150.failToRegen
	#1154 ZD0209:SimpleValve(inputOpen: #1149, inputClose: NOT #1149, statusOpen: pin 8, statusClose: pin 9, reset: pin 4, timeToOpenClose: pin 10)
	out 9 "открыть ЗДЭ02.09" <= #1154.outputOpen
	out 10 "закрыть ЗДЭ02.09" <= #1154.outputClose
	out 11 "авария открытия ЗДЭ02.09" <= #1154.errorToOpen
	out 12 "авария закрытия ЗДЭ02.09" <= #1154.errorToClose
END_MACRO
#1155 DD2_DO.6 <= #1147.out 2
#1156 regeneratedFS020103 <= #1147.out 3
#1157 filterFailToRegen020103 <= #1147.out 4
#1158 DD2_DO.20 <= #1147.out 5
#1159 DD2_DO.21 <= #1147.out 6
#1160 errorToOpenZD0203 <= #1147.out 7
#1161 errorToCloseZD0203 <= #1147.out 8
#1162 DD3_DO.0 <= #1147.out 9
#1163 DD3_DO.1 <= #1147.out 10
#1164 errorToOpenZD0209 <= #1147.out 11
#1165 errorToCloseZD0209 <= #1147.out 12
#1166 MACRO управление промывкой фильтра ФС02.01.04(pin 1 "сигнал на промывку": #1147.out 1, pin 2 "авария фильтра": DD6_DI.27, pin 3 "подтверждение промывки": DD6_DI.26, pin 4 "сброс аварий": alarmReset, pin 5 "начать очередь снова": filterStartNewQueue, pin 6 "ЗДЭ02.04 открыта": DD7_DI.22, pin 7 "ЗДЭ02.04 закрыта": DD7_DI.23, pin 8 "ЗДЭ02.10 открыта": DD8_DI.2, pin 9 "ЗДЭ02.10 закрыта": DD8_DI.3, pin 10 "время движения ЗДЭ": timeToOpenCloseValve, pin 11 "авария питания ЗДЭ02.04": DD9_DI.7, pin 12 "авария питания ЗДЭ02.10": DD9_DI.13)
	(* <- выход использовать в / последнем фильтре для / начала очереди заново *)
	(* если открыт = промывка *)
	(* если открыт = фильтрация *)
	out 1 "следующий в очереди" <= #1169.output
	out 2 "промыть ФС02.01.04" <= #1168
	#1167 ZD0204:SimpleValve(inputOpen: NOT #1168, inputClose: #1168, statusOpen: pin 6, statusClose: pin 7, reset: pin 4, timeToOpenClose: pin 10)
	out 5 "открыть ЗДЭ02.04" <= #1167.outputOpen
	out 6 "закрыть ЗДЭ02.04" <= #1167.outputClose
	out 7 "авария открытия ЗДЭ02.04" <= #1167.errorToOpen
	#1168 OR(panTestValvesFS020104, #1169.regenFilterOUT)
	out 8 "авария закрытия ЗДЭ02.04" <= #1167.errorToClose
	#1169 FS020104manager:FilterQueueManager(input: pin 1, filterAlarm: #1170, regenFilterStatus: pin 3, alarmReset: pin 4, startNextLoop: pin 5)
	#1170 OR(alarmZD020410, pin 2, pin 11, pin 12)
	#1171 OR(#1167.errorToOpen, #1167.errorToClose, #1173.errorToOpen, #1173.errorToClose)
	#1172 alarmZD020410 <= #1171
	out 3 "ФС02.01.04 промыт" <= #1169.regenerated
	out 4 "не удалось промыть" <= #1169.failToRegen
	#1173 ZD0210:SimpleValve(inputOpen: #1168, inputClose: NOT #1168, statusOpen: pin 8, statusClose: pin 9, reset: pin 4, timeToOpenClose: pin 10)
	out 9 "открыть ЗДЭ02.10" <= #1173.outputOpen
	out 10 "закрыть ЗДЭ02.10" <= #1173.outputClose
	out 11 "авария открытия ЗДЭ02.10" <= #1173.errorToOpen
	out 12 "авария закрытия ЗДЭ02.10" <= #1173.errorToClose
END_MACRO
#1174 DD2_DO.7 <= #1166.out 2
#1175 regeneratedFS020104 <= #1166.out 3
#1176 filterFailToRegen020104 <= #1166.out 4
#1177 DD2_DO.22 <= #1166.out 5
#1178 DD2_DO.23 <= #1166.out 6
#1179 errorToOpenZD0204 <= #1166.out 7
#1180 errorToCloseZD0204 <= #1166.out 8
#1181 DD3_DO.2 <= #1166.out 9
#1182 DD3_DO.3 <= #1166.out 10
#1183 errorToOpenZD0210 <= #1166.out 11
#1184 errorToCloseZD0210 <= #1166.out 12
#1185 MACRO управление промывкой фильтра ФС02.01.05(pin 1 "сигнал на промывку": #1166.out 1, pin 2 "авария фильтра": DD6_DI.29, pin 3 "подтверждение промывки": DD6_DI.28, pin 4 "сброс аварий": alarmReset, pin 5 "начать очередь снова": filterStartNewQueue, pin 6 "ЗДЭ02.05 открыта": DD7_DI.24, pin 7 "ЗДЭ02.05 закрыта": DD7_DI.25, pin 8 "ЗДЭ02.11 открыта": DD8_DI.4, pin 9 "ЗДЭ02.11 закрыта": DD8_DI.5, pin 10 "время движения ЗДЭ": timeToOpenCloseValve, pin 11 "авария питания ЗДЭ02.05": DD9_DI.8, pin 12 "авария питания ЗДЭ02.11": DD9_DI.14)
	(* <- выход использовать в / последнем фильтре для / начала очереди заново *)
	(* если открыт = промывка *)
	(* если открыт = фильтрация *)
	out 1 "следующий в очереди" <= #1188.output
	out 2 "промыть ФС02.01.05" <= #1187
	#1186 ZD0205:SimpleValve(inputOpen: NOT #1187, inputClose: #1187, statusOpen: pin 6, statusClose: pin 7, reset: pin 4, timeToOpenClose: pin 10)
	out 5 "открыть ЗДЭ02.05" <= #1186.outputOpen
	out 6 "закрыть ЗДЭ02.05" <= #1186.outputClose
	out 7 "авария открытия ЗДЭ02.05" <= #1186.errorToOpen
	#1187 OR(panTestValvesFS020105, #1188.regenFilterOUT)
	out 8 "авария закрытия ЗДЭ02.05" <= #1186.errorToClose
	#1188 FS020105manager:FilterQueueManager(input: pin 1, filterAlarm: #1189, regenFilterStatus: pin 3, alarmReset: pin 4, startNextLoop: pin 5)
	#1189 OR(alarmZD020511, pin 2, pin 11, pin 12)
	#1190 OR(#1186.errorToOpen, #1186.errorToClose, #1192.errorToOpen, #1192.errorToClose)
	#1191 alarmZD020511 <= #1190
	out 3 "ФС02.01.05 промыт" <= #1188.regenerated
	out 4 "не удалось промыть" <= #1188.failToRegen
	#1192 ZD0211:SimpleValve(inputOpen: #1187, inputClose: NOT #1187, statusOpen: pin 8, statusClose: pin 9, reset: pin 4, timeToOpenClose: pin 10)
	out 9 "открыть ЗДЭ02.11" <= #1192.outputOpen
	out 10 "закрыть ЗДЭ02.11" <= #1192.outputClose
	out 11 "авария открытия ЗДЭ02.11" <= #1192.errorToOpen
	out 12 "авария закрытия ЗДЭ02.11" <= #1192.errorToClose
END_MACRO
#1193 DD2_DO.8 <= #1185.out 2
#1194 regeneratedFS020105 <= #1185.out 3
#1195 filterFailToRegen020105 <= #1185.out 4
#1196 DD2_DO.24 <= #1185.out 5
#1197 DD2_DO.25 <= #1185.out 6
#1198 errorToOpenZD0205 <= #1185.out 7
#1199 errorToCloseZD0205 <= #1185.out 8
#1200 DD3_DO.4 <= #1185.out 9
#1201 DD3_DO.5 <= #1185.out 10
#1202 errorToOpenZD0211 <= #1185.out 11
#1203 errorToCloseZD0211 <= #1185.out 12
#1204 MACRO управление промывкой фильтра ФС02.01.06(pin 1 "сигнал на промывку": #1185.out 1, pin 2 "авария фильтра": DD6_DI.31, pin 3 "подтверждение промывки": DD6_DI.30, pin 4 "сброс аварий": alarmReset, pin 5 "начать очередь снова": filterStartNewQueue, pin 6 "ЗДЭ02.06 открыта": DD7_DI.26, pin 7 "ЗДЭ02.06 закрыта": DD7_DI.27, pin 8 "ЗДЭ02.12 открыта": DD8_DI.6, pin 9 "ЗДЭ02.12 закрыта": DD8_DI.7, pin 10 "время движения ЗДЭ": timeToOpenCloseValve, pin 11 "авария питания ЗДЭ02.06": DD9_DI.9, pin 12 "авария питания ЗДЭ02.12": DD9_DI.15)
	(* <- выход использовать в / последнем фильтре для / начала очереди заново *)
	(* если открыт = промывка *)
	(* если открыт = фильтрация *)
	out 1 "следующий в очереди" <= #1207.output
	out 2 "промыть ФС02.01.06" <= #1206
	#1205 ZD0206:SimpleValve(inputOpen: NOT #1206, inputClose: #1206, statusOpen: pin 6, statusClose: pin 7, reset: pin 4, timeToOpenClose: pin 10)
	out 5 "открыть ЗДЭ02.06" <= #1205.outputOpen
	out 6 "закрыть ЗДЭ02.06" <= #1205.outputClose
	out 7 "авария открытия ЗДЭ02.06" <= #1205.errorToOpen
	#1206 OR(panTestValvesFS020106, #1207.regenFilterOUT)
	out 8 "авария закрытия ЗДЭ02.06" <= #1205.errorToClose
	#1207 FS020106manager:FilterQueueManager(input: pin 1, filterAlarm: #1208, regenFilterStatus: pin 3, alarmReset: pin 4, startNextLoop: pin 5)
	#1208 OR(alarmZD020612, pin 2, pin 11, pin 12)
	#1209 OR(#1205.errorToOpen, #1205.errorToClose, #1211.errorToOpen, #1211.errorToClose)
	#1210 alarmZD020612 <= #1209
	out 3 "ФС02.01.06 промыт" <= #1207.regenerated
	out 4 "не удалось промыть" <= #1207.failToRegen
	#1211 ZD0212:SimpleValve(inputOpen: #1206, inputClose: NOT #1206, statusOpen: pin 8, statusClose: pin 9, reset: pin 4, timeToOpenClose: pin 10)
	out 9 "открыть ЗДЭ02.12" <= #1211.outputOpen
	out 10 "закрыть ЗДЭ02.12" <= #1211.outputClose
	out 11 "авария открытия ЗДЭ02.12" <= #1211.errorToOpen
	out 12 "авария закрытия ЗДЭ02.12" <= #1211.errorToClose
END_MACRO
#1212 DD2_DO.9 <= #1204.out 2
#1213 regeneratedFS020106 <= #1204.out 3
#1214 filterFailToRegen020106 <= #1204.out 4
#1215 DD2_DO.26 <= #1204.out 5
#1216 DD2_DO.27 <= #1204.out 6
#1217 errorToOpenZD0206 <= #1204.out 7
#1218 errorToCloseZD0206 <= #1204.out 8
#1219 DD3_DO.6 <= #1204.out 9
#1220 DD3_DO.7 <= #1204.out 10
#1221 errorToOpenZD0212 <= #1204.out 11
#1222 errorToCloseZD0212 <= #1204.out 12
#1223 MACRO управление промывкой фильтра ФС02.02.01(pin 1 "сигнал на промывку": #1204.out 1, pin 2 "авария фильтра": DD7_DI.1, pin 3 "подтверждение промывки": DD7_DI.0, pin 4 "сброс аварий": alarmReset, pin 5 "начать очередь снова": filterStartNewQueue, pin 6 "ЗДЭ02.13 открыта": DD8_DI.8, pin 7 "ЗДЭ02.13 закрыта": DD8_DI.9, pin 8 "ЗДЭ02.19 открыта": DD8_DI.20, pin 9 "ЗДЭ02.19 закрыта": DD8_DI.21, pin 10 "время движения ЗДЭ": timeToOpenCloseValve, pin 11 "авария питания ЗДЭ02.13": DD9_DI.16, pin 12 "авария питания ЗДЭ02.19": DD9_DI.22)
	(* <- выход использовать в / последнем фильтре для / начала очереди заново *)
	(* если открыт = промывка *)
	(* если открыт = фильтрация *)
	out 1 "следующий в очереди" <= #1226.output
	out 2 "промыть ФС02.02.01" <= #1225
	#1224 ZD0213:SimpleValve(inputOpen: NOT #1225, inputClose: #1225, statusOpen: pin 6, statusClose: pin 7, reset: pin 4, timeToOpenClose: pin 10)
	out 5 "открыть ЗДЭ02.13" <= #1224.outputOpen
	out 6 "закрыть ЗДЭ02.13" <= #1224.outputClose
	out 7 "авария открытия ЗДЭ02.13" <= #1224.errorToOpen
	#1225 OR(panTestValvesFS020201, #1226.regenFilterOUT)
	out 8 "авария закрытия ЗДЭ02.13" <= #1224.errorToClose
	#1226 FS020201manager:FilterQueueManager(input: pin 1, filterAlarm: #1227, regenFilterStatus: pin 3, alarmReset: pin 4, startNextLoop: pin 5)
	#1227 OR(alarmZD021319, pin 2, pin 11, pin 12)
	#1228 OR(#1224.errorToOpen, #1224.errorToClose, #1230.errorToOpen, #1230.errorToClose)
	#1229 alarmZD021319 <= #1228
	out 3 "ФС02.02.01 промыт" <= #1226.regenerated
